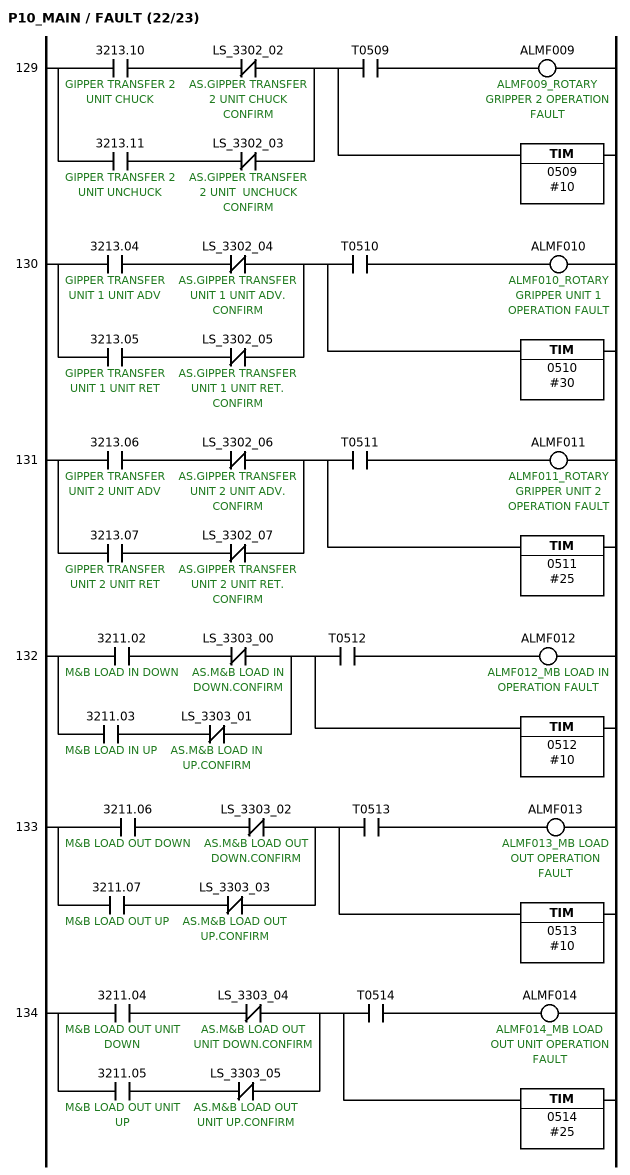
; [picture p24: P10_MAIN / FAULT, rungs 129-134]
; rung 129
LD 3213.10  ; GIPPER TRANSFER 2 UNIT CHUCK
ANDNOT LS_3302_02  ; AS.GIPPER TRANSFER 2 UNIT CHUCK CONFIRM
LD 3213.11  ; GIPPER TRANSFER 2 UNIT UNCHUCK
ANDNOT LS_3302_03  ; AS.GIPPER TRANSFER 2 UNIT  UNCHUCK CONFIRM
ORLD
OUT TR0
AND T0509
OUT ALMF009  ; ALMF009_ROTARY GRIPPER 2 OPERATION FAULT
LD TR0
TIM 0509 #10
; rung 130
LD 3213.04  ; GIPPER TRANSFER UNIT 1 UNIT ADV
ANDNOT LS_3302_04  ; AS.GIPPER TRANSFER UNIT 1 UNIT ADV. CONFIRM
LD 3213.05  ; GIPPER TRANSFER UNIT 1 UNIT RET
ANDNOT LS_3302_05  ; AS.GIPPER TRANSFER UNIT 1 UNIT RET. CONFIRM
ORLD
OUT TR0
AND T0510
OUT ALMF010  ; ALMF010_ROTARY GRIPPER UNIT 1 OPERATION FAULT
LD TR0
TIM 0510 #30
; rung 131
LD 3213.06  ; GIPPER TRANSFER UNIT 2 UNIT ADV
ANDNOT LS_3302_06  ; AS.GIPPER TRANSFER UNIT 2 UNIT ADV. CONFIRM
LD 3213.07  ; GIPPER TRANSFER UNIT 2 UNIT RET
ANDNOT LS_3302_07  ; AS.GIPPER TRANSFER UNIT 2 UNIT RET. CONFIRM
ORLD
OUT TR0
AND T0511
OUT ALMF011  ; ALMF011_ROTARY GRIPPER UNIT 2 OPERATION FAULT
LD TR0
TIM 0511 #25
; rung 132
LD 3211.02  ; M&B LOAD IN DOWN
ANDNOT LS_3303_00  ; AS.M&B LOAD IN DOWN.CONFIRM
LD 3211.03  ; M&B LOAD IN UP
ANDNOT LS_3303_01  ; AS.M&B LOAD IN UP.CONFIRM
ORLD
OUT TR0
AND T0512
OUT ALMF012  ; ALMF012_MB LOAD IN OPERATION FAULT
LD TR0
TIM 0512 #10
; rung 133
LD 3211.06  ; M&B LOAD OUT DOWN
ANDNOT LS_3303_02  ; AS.M&B LOAD OUT DOWN.CONFIRM
LD 3211.07  ; M&B LOAD OUT UP
ANDNOT LS_3303_03  ; AS.M&B LOAD OUT UP.CONFIRM
ORLD
OUT TR0
AND T0513
OUT ALMF013  ; ALMF013_MB LOAD OUT OPERATION FAULT
LD TR0
TIM 0513 #10
; rung 134
LD 3211.04  ; M&B LOAD OUT UNIT DOWN
ANDNOT LS_3303_04  ; AS.M&B LOAD OUT UNIT DOWN.CONFIRM
LD 3211.05  ; M&B LOAD OUT UNIT UP
ANDNOT LS_3303_05  ; AS.M&B LOAD OUT UNIT UP.CONFIRM
ORLD
OUT TR0
AND T0514
OUT ALMF014  ; ALMF014_MB LOAD OUT UNIT OPERATION FAULT
LD TR0
TIM 0514 #25

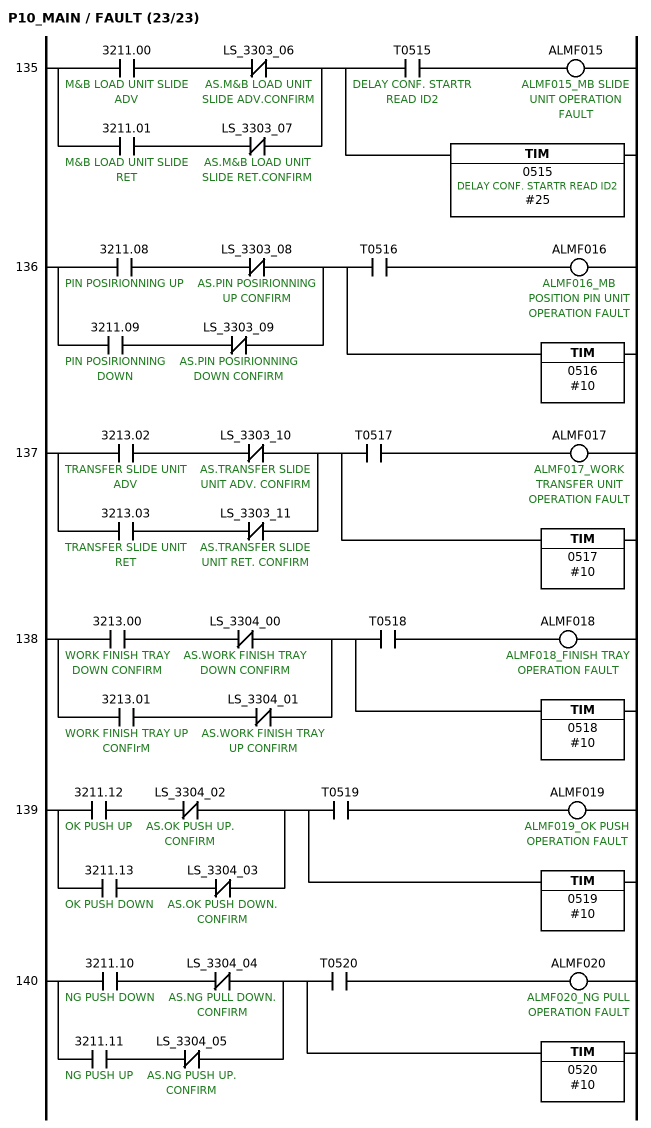
; rung 135
LD 3211.00  ; M&B LOAD UNIT SLIDE ADV
ANDNOT LS_3303_06  ; AS.M&B LOAD UNIT SLIDE ADV.CONFIRM
LD 3211.01  ; M&B LOAD UNIT SLIDE RET
ANDNOT LS_3303_07  ; AS.M&B LOAD UNIT SLIDE RET.CONFIRM
ORLD
OUT TR0
AND T0515  ; DELAY CONF. STARTR READ ID2
OUT ALMF015  ; ALMF015_MB SLIDE UNIT OPERATION FAULT
LD TR0
TIM 0515 #25  ; DELAY CONF. STARTR READ ID2
; rung 136
LD 3211.08  ; PIN POSIRIONNING UP
ANDNOT LS_3303_08  ; AS.PIN POSIRIONNING UP CONFIRM
LD 3211.09  ; PIN POSIRIONNING DOWN
ANDNOT LS_3303_09  ; AS.PIN POSIRIONNING DOWN CONFIRM
ORLD
OUT TR0
AND T0516
OUT ALMF016  ; ALMF016_MB POSITION PIN UNIT OPERATION FAULT
LD TR0
TIM 0516 #10
; rung 137
LD 3213.02  ; TRANSFER SLIDE UNIT ADV
ANDNOT LS_3303_10  ; AS.TRANSFER SLIDE UNIT ADV. CONFIRM
LD 3213.03  ; TRANSFER SLIDE UNIT RET
ANDNOT LS_3303_11  ; AS.TRANSFER SLIDE UNIT RET. CONFIRM
ORLD
OUT TR0
AND T0517
OUT ALMF017  ; ALMF017_WORK TRANSFER UNIT OPERATION FAULT
LD TR0
TIM 0517 #10
; rung 138
LD 3213.00  ; WORK FINISH TRAY DOWN CONFIRM
ANDNOT LS_3304_00  ; AS.WORK FINISH TRAY DOWN CONFIRM
LD 3213.01  ; WORK FINISH TRAY UP CONFIrM
ANDNOT LS_3304_01  ; AS.WORK FINISH TRAY UP CONFIRM
ORLD
OUT TR0
AND T0518
OUT ALMF018  ; ALMF018_FINISH TRAY OPERATION FAULT
LD TR0
TIM 0518 #10
; rung 139
LD 3211.12  ; OK PUSH UP
ANDNOT LS_3304_02  ; AS.OK PUSH UP. CONFIRM
LD 3211.13  ; OK PUSH DOWN
ANDNOT LS_3304_03  ; AS.OK PUSH DOWN. CONFIRM
ORLD
OUT TR0
AND T0519
OUT ALMF019  ; ALMF019_OK PUSH OPERATION FAULT
LD TR0
TIM 0519 #10
; rung 140
LD 3211.10  ; NG PUSH DOWN
ANDNOT LS_3304_04  ; AS.NG PULL DOWN. CONFIRM
LD 3211.11  ; NG PUSH UP
ANDNOT LS_3304_05  ; AS.NG PUSH UP. CONFIRM
ORLD
OUT TR0
AND T0520
OUT ALMF020  ; ALMF020_NG PULL OPERATION FAULT
LD TR0
TIM 0520 #10

### Section INPUT

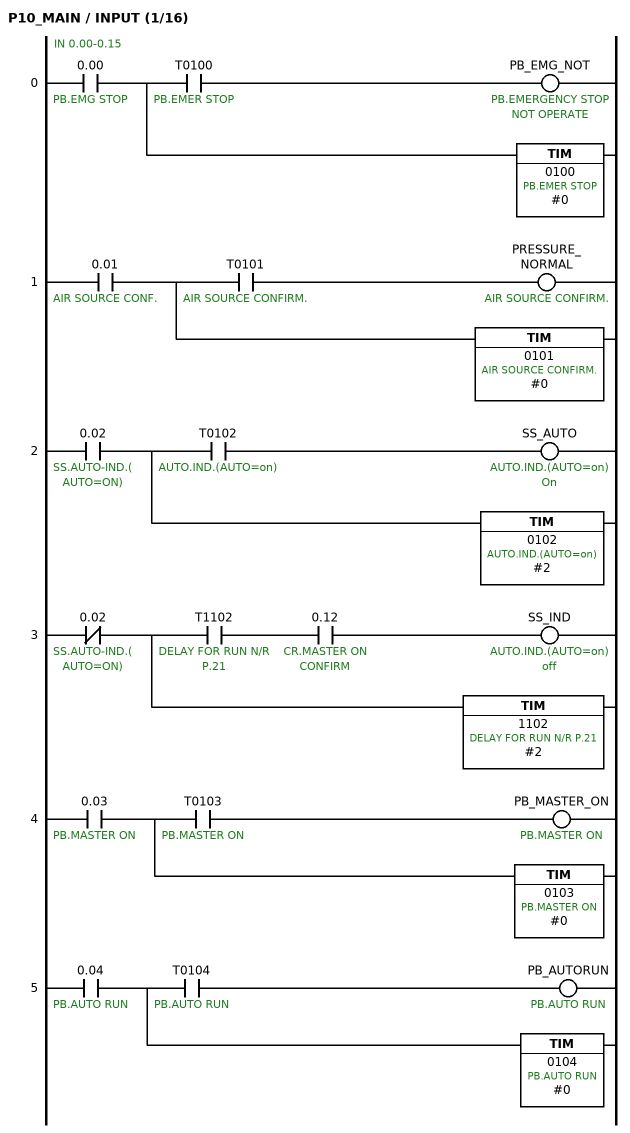
; rung 0: IN 0.00-0.15
LD 0.00  ; PB.EMG STOP
OUT TR0
AND T0100  ; PB.EMER STOP
OUT PB_EMG_NOT  ; PB.EMERGENCY STOP NOT OPERATE
LD TR0
TIM 0100 #0  ; PB.EMER STOP
; rung 1
LD 0.01  ; AIR SOURCE CONF.
OUT TR0
AND T0101  ; AIR SOURCE CONFIRM.
OUT PRESSURE_NORMAL  ; AIR SOURCE CONFIRM.
LD TR0
TIM 0101 #0  ; AIR SOURCE CONFIRM.
; rung 2
LD 0.02  ; SS.AUTO-IND.(AUTO=ON)
OUT TR0
AND T0102  ; AUTO.IND.(AUTO=on)
OUT SS_AUTO  ; AUTO.IND.(AUTO=on) On
LD TR0
TIM 0102 #2  ; AUTO.IND.(AUTO=on)
; rung 3
LDNOT 0.02  ; SS.AUTO-IND.(AUTO=ON)
OUT TR0
AND T1102  ; DELAY FOR RUN N/R P.21
AND 0.12  ; CR.MASTER ON CONFIRM
OUT SS_IND  ; AUTO.IND.(AUTO=on) off
LD TR0
TIM 1102 #2  ; DELAY FOR RUN N/R P.21
; rung 4
LD 0.03  ; PB.MASTER ON
OUT TR0
AND T0103  ; PB.MASTER ON
OUT PB_MASTER_ON  ; PB.MASTER ON
LD TR0
TIM 0103 #0  ; PB.MASTER ON
; rung 5
LD 0.04  ; PB.AUTO RUN
OUT TR0
AND T0104  ; PB.AUTO RUN
OUT PB_AUTORUN  ; PB.AUTO RUN
LD TR0
TIM 0104 #0  ; PB.AUTO RUN

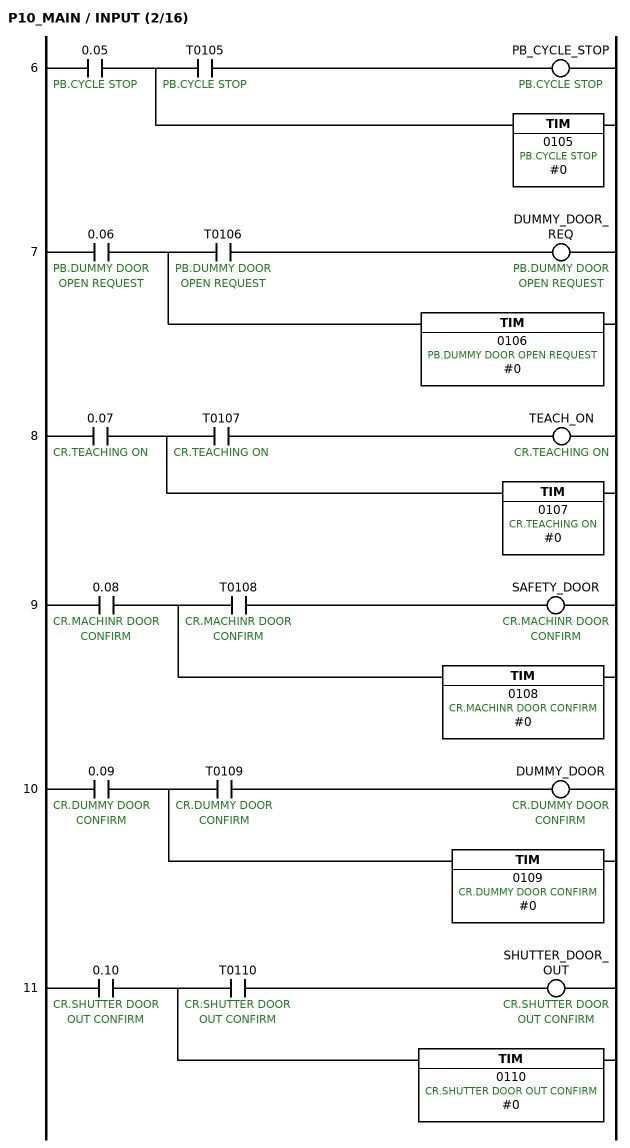
; rung 6
LD 0.05  ; PB.CYCLE STOP
OUT TR0
AND T0105  ; PB.CYCLE STOP
OUT PB_CYCLE_STOP  ; PB.CYCLE STOP
LD TR0
TIM 0105 #0  ; PB.CYCLE STOP
; rung 7
LD 0.06  ; PB.DUMMY DOOR OPEN REQUEST
OUT TR0
AND T0106  ; PB.DUMMY DOOR OPEN REQUEST
OUT DUMMY_DOOR_REQ  ; PB.DUMMY DOOR OPEN REQUEST
LD TR0
TIM 0106 #0  ; PB.DUMMY DOOR OPEN REQUEST
; rung 8
LD 0.07  ; CR.TEACHING ON
OUT TR0
AND T0107  ; CR.TEACHING ON
OUT TEACH_ON  ; CR.TEACHING ON
LD TR0
TIM 0107 #0  ; CR.TEACHING ON
; rung 9
LD 0.08  ; CR.MACHINR DOOR CONFIRM
OUT TR0
AND T0108  ; CR.MACHINR DOOR CONFIRM
OUT SAFETY_DOOR  ; CR.MACHINR DOOR CONFIRM
LD TR0
TIM 0108 #0  ; CR.MACHINR DOOR CONFIRM
; rung 10
LD 0.09  ; CR.DUMMY DOOR CONFIRM
OUT TR0
AND T0109  ; CR.DUMMY DOOR CONFIRM
OUT DUMMY_DOOR  ; CR.DUMMY DOOR CONFIRM
LD TR0
TIM 0109 #0  ; CR.DUMMY DOOR CONFIRM
; rung 11
LD 0.10  ; CR.SHUTTER DOOR OUT CONFIRM
OUT TR0
AND T0110  ; CR.SHUTTER DOOR OUT CONFIRM
OUT SHUTTER_DOOR_OUT  ; CR.SHUTTER DOOR OUT CONFIRM
LD TR0
TIM 0110 #0  ; CR.SHUTTER DOOR OUT CONFIRM

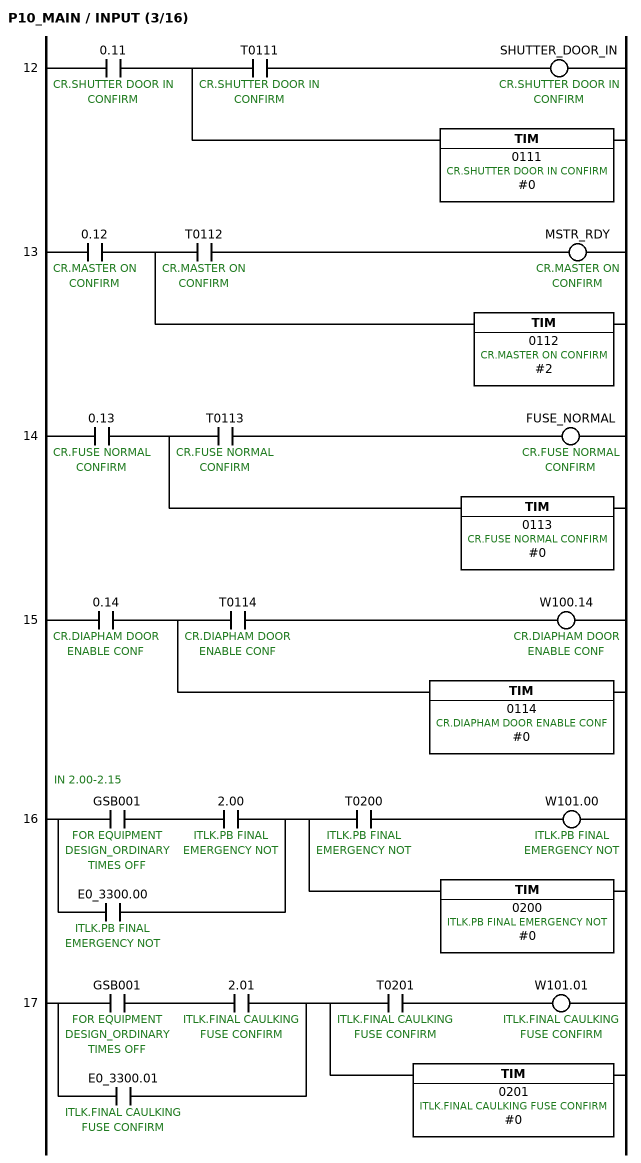
; rung 12
LD 0.11  ; CR.SHUTTER DOOR IN CONFIRM
OUT TR0
AND T0111  ; CR.SHUTTER DOOR IN CONFIRM
OUT SHUTTER_DOOR_IN  ; CR.SHUTTER DOOR IN CONFIRM
LD TR0
TIM 0111 #0  ; CR.SHUTTER DOOR IN CONFIRM
; rung 13
LD 0.12  ; CR.MASTER ON CONFIRM
OUT TR0
AND T0112  ; CR.MASTER ON CONFIRM
OUT MSTR_RDY  ; CR.MASTER ON CONFIRM
LD TR0
TIM 0112 #2  ; CR.MASTER ON CONFIRM
; rung 14
LD 0.13  ; CR.FUSE NORMAL CONFIRM
OUT TR0
AND T0113  ; CR.FUSE NORMAL CONFIRM
OUT FUSE_NORMAL  ; CR.FUSE NORMAL CONFIRM
LD TR0
TIM 0113 #0  ; CR.FUSE NORMAL CONFIRM
; rung 15
LD 0.14  ; CR.DIAPHAM DOOR ENABLE CONF
OUT TR0
AND T0114  ; CR.DIAPHAM DOOR ENABLE CONF
OUT W100.14  ; CR.DIAPHAM DOOR ENABLE CONF
LD TR0
TIM 0114 #0  ; CR.DIAPHAM DOOR ENABLE CONF
; rung 16: IN 2.00-2.15
LD GSB001  ; FOR EQUIPMENT DESIGN_ORDINARY TIMES OFF
AND 2.00  ; ITLK.PB FINAL EMERGENCY NOT
OR E0_3300.00  ; ITLK.PB FINAL EMERGENCY NOT
OUT TR0
AND T0200  ; ITLK.PB FINAL EMERGENCY NOT
OUT W101.00  ; ITLK.PB FINAL EMERGENCY NOT
LD TR0
TIM 0200 #0  ; ITLK.PB FINAL EMERGENCY NOT
; rung 17
LD GSB001  ; FOR EQUIPMENT DESIGN_ORDINARY TIMES OFF
AND 2.01  ; ITLK.FINAL CAULKING FUSE CONFIRM
OR E0_3300.01  ; ITLK.FINAL CAULKING FUSE CONFIRM
OUT TR0
AND T0201  ; ITLK.FINAL CAULKING FUSE CONFIRM
OUT W101.01  ; ITLK.FINAL CAULKING FUSE CONFIRM
LD TR0
TIM 0201 #0  ; ITLK.FINAL CAULKING FUSE CONFIRM

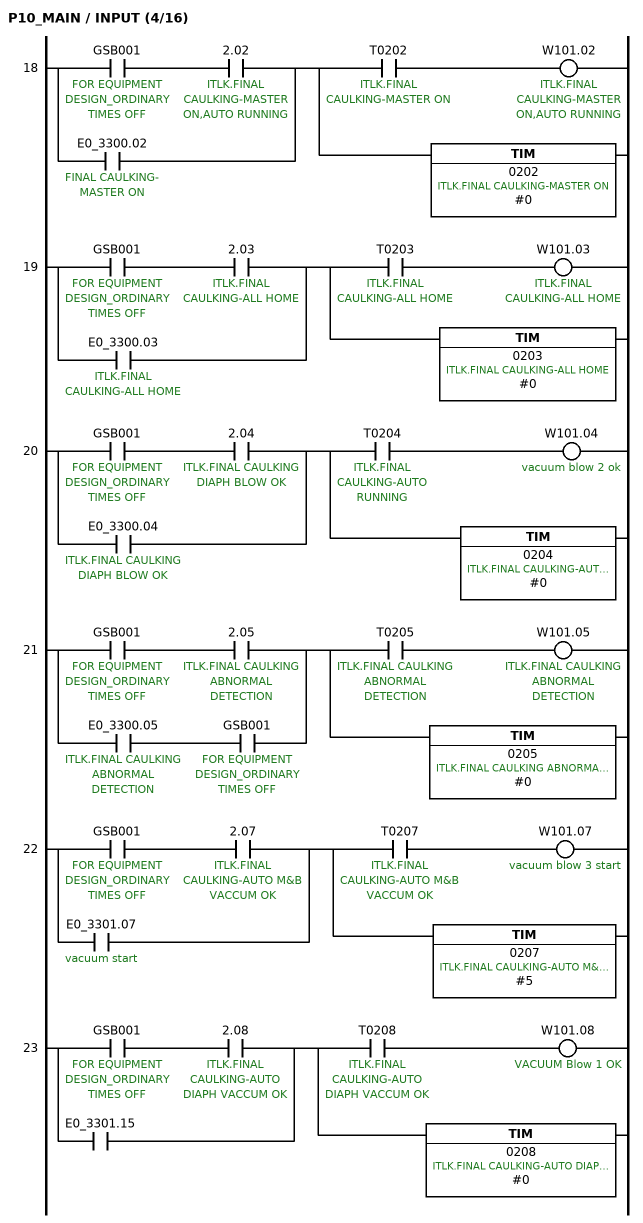
; rung 18
LD GSB001  ; FOR EQUIPMENT DESIGN_ORDINARY TIMES OFF
AND 2.02  ; ITLK.FINAL CAULKING-MASTER ON,AUTO RUNNING
OR E0_3300.02  ; FINAL CAULKING-MASTER ON
OUT TR0
AND T0202  ; ITLK.FINAL CAULKING-MASTER ON
OUT W101.02  ; ITLK.FINAL CAULKING-MASTER ON,AUTO RUNNING
LD TR0
TIM 0202 #0  ; ITLK.FINAL CAULKING-MASTER ON
; rung 19
LD GSB001  ; FOR EQUIPMENT DESIGN_ORDINARY TIMES OFF
AND 2.03  ; ITLK.FINAL CAULKING-ALL HOME
OR E0_3300.03  ; ITLK.FINAL CAULKING-ALL HOME
OUT TR0
AND T0203  ; ITLK.FINAL CAULKING-ALL HOME
OUT W101.03  ; ITLK.FINAL CAULKING-ALL HOME
LD TR0
TIM 0203 #0  ; ITLK.FINAL CAULKING-ALL HOME
; rung 20
LD GSB001  ; FOR EQUIPMENT DESIGN_ORDINARY TIMES OFF
AND 2.04  ; ITLK.FINAL CAULKING DIAPH BLOW OK
OR E0_3300.04  ; ITLK.FINAL CAULKING DIAPH BLOW OK
OUT TR0
AND T0204  ; ITLK.FINAL CAULKING-AUTO RUNNING
OUT W101.04  ; vacuum blow 2 ok
LD TR0
TIM 0204 #0  ; ITLK.FINAL CAULKING-AUTO RUNNING
; rung 21
LD GSB001  ; FOR EQUIPMENT DESIGN_ORDINARY TIMES OFF
AND 2.05  ; ITLK.FINAL CAULKING ABNORMAL DETECTION
LD E0_3300.05  ; ITLK.FINAL CAULKING ABNORMAL DETECTION
AND GSB001  ; FOR EQUIPMENT DESIGN_ORDINARY TIMES OFF
ORLD
OUT TR0
AND T0205  ; ITLK.FINAL CAULKING ABNORMAL DETECTION
OUT W101.05  ; ITLK.FINAL CAULKING ABNORMAL DETECTION
LD TR0
TIM 0205 #0  ; ITLK.FINAL CAULKING ABNORMAL DETECTION
; rung 22
LD GSB001  ; FOR EQUIPMENT DESIGN_ORDINARY TIMES OFF
AND 2.07  ; ITLK.FINAL CAULKING-AUTO M&B VACCUM OK
OR E0_3301.07  ; vacuum start
OUT TR0
AND T0207  ; ITLK.FINAL CAULKING-AUTO M&B VACCUM OK
OUT W101.07  ; vacuum blow 3 start
LD TR0
TIM 0207 #5  ; ITLK.FINAL CAULKING-AUTO M&B VACCUM OK
; rung 23
LD GSB001  ; FOR EQUIPMENT DESIGN_ORDINARY TIMES OFF
AND 2.08  ; ITLK.FINAL CAULKING-AUTO DIAPH VACCUM OK
OR E0_3301.15
OUT TR0
AND T0208  ; ITLK.FINAL CAULKING-AUTO DIAPH VACCUM OK
OUT W101.08  ; VACUUM Blow 1 OK
LD TR0
TIM 0208 #0  ; ITLK.FINAL CAULKING-AUTO DIAPH VACCUM OK

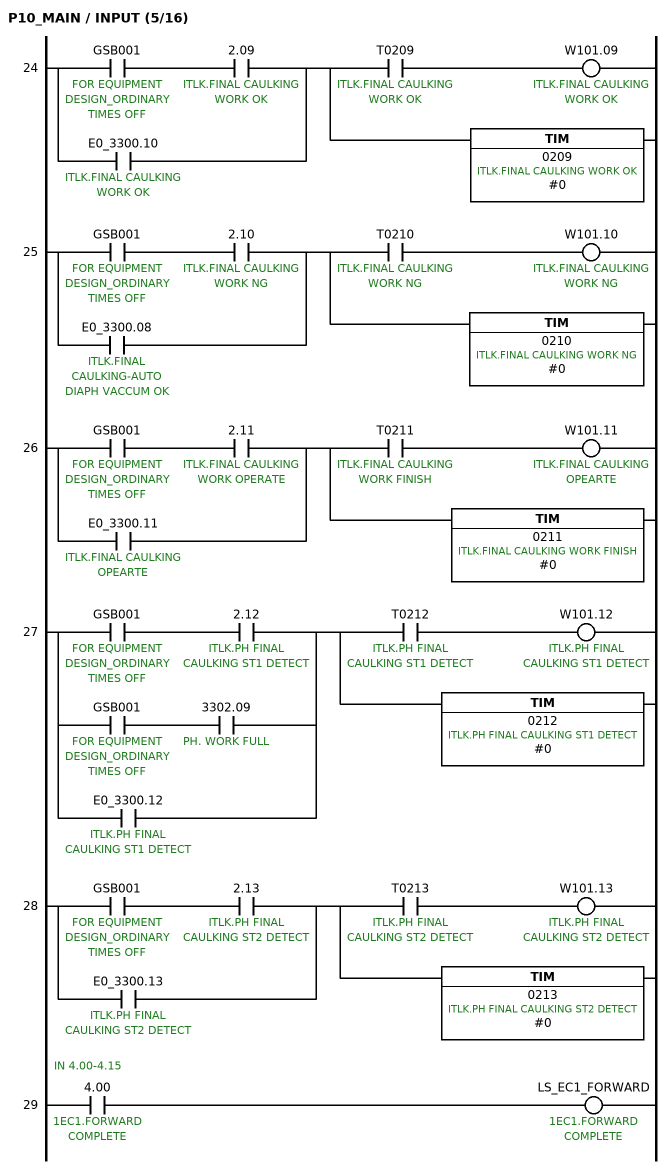
; rung 24
LD GSB001  ; FOR EQUIPMENT DESIGN_ORDINARY TIMES OFF
AND 2.09  ; ITLK.FINAL CAULKING WORK OK
OR E0_3300.10  ; ITLK.FINAL CAULKING WORK OK
OUT TR0
AND T0209  ; ITLK.FINAL CAULKING WORK OK
OUT W101.09  ; ITLK.FINAL CAULKING WORK OK
LD TR0
TIM 0209 #0  ; ITLK.FINAL CAULKING WORK OK
; rung 25
LD GSB001  ; FOR EQUIPMENT DESIGN_ORDINARY TIMES OFF
AND 2.10  ; ITLK.FINAL CAULKING WORK NG
OR E0_3300.08  ; ITLK.FINAL CAULKING-AUTO DIAPH VACCUM OK
OUT TR0
AND T0210  ; ITLK.FINAL CAULKING WORK NG
OUT W101.10  ; ITLK.FINAL CAULKING WORK NG
LD TR0
TIM 0210 #0  ; ITLK.FINAL CAULKING WORK NG
; rung 26
LD GSB001  ; FOR EQUIPMENT DESIGN_ORDINARY TIMES OFF
AND 2.11  ; ITLK.FINAL CAULKING WORK OPERATE
OR E0_3300.11  ; ITLK.FINAL CAULKING OPEARTE
OUT TR0
AND T0211  ; ITLK.FINAL CAULKING WORK FINISH
OUT W101.11  ; ITLK.FINAL CAULKING OPEARTE
LD TR0
TIM 0211 #0  ; ITLK.FINAL CAULKING WORK FINISH
; rung 27
LD GSB001  ; FOR EQUIPMENT DESIGN_ORDINARY TIMES OFF
AND 2.12  ; ITLK.PH FINAL CAULKING ST1 DETECT
LD GSB001  ; FOR EQUIPMENT DESIGN_ORDINARY TIMES OFF
AND 3302.09  ; PH. WORK FULL
ORLD
OR E0_3300.12  ; ITLK.PH FINAL CAULKING ST1 DETECT
OUT TR0
AND T0212  ; ITLK.PH FINAL CAULKING ST1 DETECT
OUT W101.12  ; ITLK.PH FINAL CAULKING ST1 DETECT
LD TR0
TIM 0212 #0  ; ITLK.PH FINAL CAULKING ST1 DETECT
; rung 28
LD GSB001  ; FOR EQUIPMENT DESIGN_ORDINARY TIMES OFF
AND 2.13  ; ITLK.PH FINAL CAULKING ST2 DETECT
OR E0_3300.13  ; ITLK.PH FINAL CAULKING ST2 DETECT
OUT TR0
AND T0213  ; ITLK.PH FINAL CAULKING ST2 DETECT
OUT W101.13  ; ITLK.PH FINAL CAULKING ST2 DETECT
LD TR0
TIM 0213 #0  ; ITLK.PH FINAL CAULKING ST2 DETECT
; rung 29: IN 4.00-4.15
LD 4.00  ; 1EC1.FORWARD COMPLETE
OUT LS_EC1_FORWARD  ; 1EC1.FORWARD COMPLETE

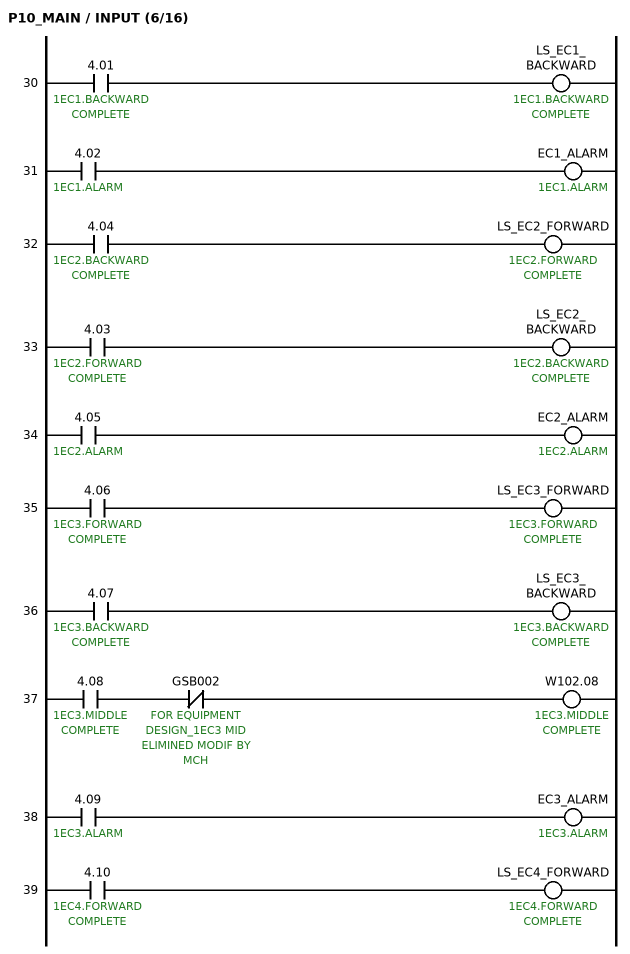
; rung 30
LD 4.01  ; 1EC1.BACKWARD COMPLETE
OUT LS_EC1_BACKWARD  ; 1EC1.BACKWARD COMPLETE
; rung 31
LD 4.02  ; 1EC1.ALARM
OUT EC1_ALARM  ; 1EC1.ALARM
; rung 32
LD 4.04  ; 1EC2.BACKWARD COMPLETE
OUT LS_EC2_FORWARD  ; 1EC2.FORWARD COMPLETE
; rung 33
LD 4.03  ; 1EC2.FORWARD COMPLETE
OUT LS_EC2_BACKWARD  ; 1EC2.BACKWARD COMPLETE
; rung 34
LD 4.05  ; 1EC2.ALARM
OUT EC2_ALARM  ; 1EC2.ALARM
; rung 35
LD 4.06  ; 1EC3.FORWARD COMPLETE
OUT LS_EC3_FORWARD  ; 1EC3.FORWARD COMPLETE
; rung 36
LD 4.07  ; 1EC3.BACKWARD COMPLETE
OUT LS_EC3_BACKWARD  ; 1EC3.BACKWARD COMPLETE
; rung 37
LD 4.08  ; 1EC3.MIDDLE COMPLETE
ANDNOT GSB002  ; FOR EQUIPMENT DESIGN_1EC3 MID ELIMINED MODIF BY MCH
OUT W102.08  ; 1EC3.MIDDLE COMPLETE
; rung 38
LD 4.09  ; 1EC3.ALARM
OUT EC3_ALARM  ; 1EC3.ALARM
; rung 39
LD 4.10  ; 1EC4.FORWARD COMPLETE
OUT LS_EC4_FORWARD  ; 1EC4.FORWARD COMPLETE

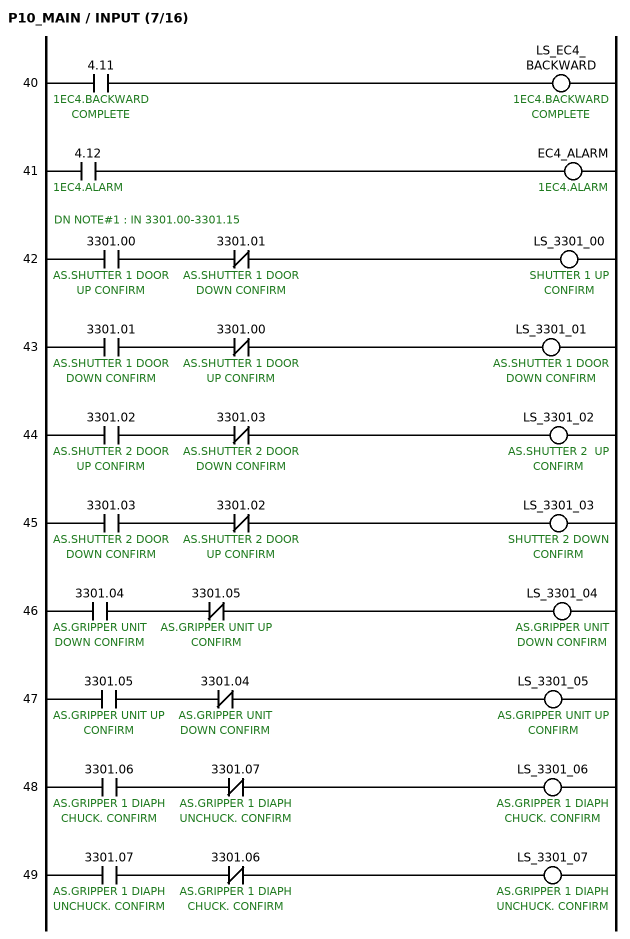
; rung 40
LD 4.11  ; 1EC4.BACKWARD COMPLETE
OUT LS_EC4_BACKWARD  ; 1EC4.BACKWARD COMPLETE
; rung 41
LD 4.12  ; 1EC4.ALARM
OUT EC4_ALARM  ; 1EC4.ALARM
; rung 42: DN NOTE#1 : IN 3301.00-3301.15
LD 3301.00  ; AS.SHUTTER 1 DOOR UP CONFIRM
ANDNOT 3301.01  ; AS.SHUTTER 1 DOOR DOWN CONFIRM
OUT LS_3301_00  ; SHUTTER 1 UP CONFIRM
; rung 43
LD 3301.01  ; AS.SHUTTER 1 DOOR DOWN CONFIRM
ANDNOT 3301.00  ; AS.SHUTTER 1 DOOR UP CONFIRM
OUT LS_3301_01  ; AS.SHUTTER 1 DOOR DOWN CONFIRM
; rung 44
LD 3301.02  ; AS.SHUTTER 2 DOOR UP CONFIRM
ANDNOT 3301.03  ; AS.SHUTTER 2 DOOR DOWN CONFIRM
OUT LS_3301_02  ; AS.SHUTTER 2  UP CONFIRM
; rung 45
LD 3301.03  ; AS.SHUTTER 2 DOOR DOWN CONFIRM
ANDNOT 3301.02  ; AS.SHUTTER 2 DOOR UP CONFIRM
OUT LS_3301_03  ; SHUTTER 2 DOWN CONFIRM
; rung 46
LD 3301.04  ; AS.GRIPPER UNIT DOWN CONFIRM
ANDNOT 3301.05  ; AS.GRIPPER UNIT UP CONFIRM
OUT LS_3301_04  ; AS.GRIPPER UNIT DOWN CONFIRM
; rung 47
LD 3301.05  ; AS.GRIPPER UNIT UP CONFIRM
ANDNOT 3301.04  ; AS.GRIPPER UNIT DOWN CONFIRM
OUT LS_3301_05  ; AS.GRIPPER UNIT UP CONFIRM
; rung 48
LD 3301.06  ; AS.GRIPPER 1 DIAPH CHUCK. CONFIRM
ANDNOT 3301.07  ; AS.GRIPPER 1 DIAPH UNCHUCK. CONFIRM
OUT LS_3301_06  ; AS.GRIPPER 1 DIAPH CHUCK. CONFIRM
; rung 49
LD 3301.07  ; AS.GRIPPER 1 DIAPH UNCHUCK. CONFIRM
ANDNOT 3301.06  ; AS.GRIPPER 1 DIAPH CHUCK. CONFIRM
OUT LS_3301_07  ; AS.GRIPPER 1 DIAPH UNCHUCK. CONFIRM

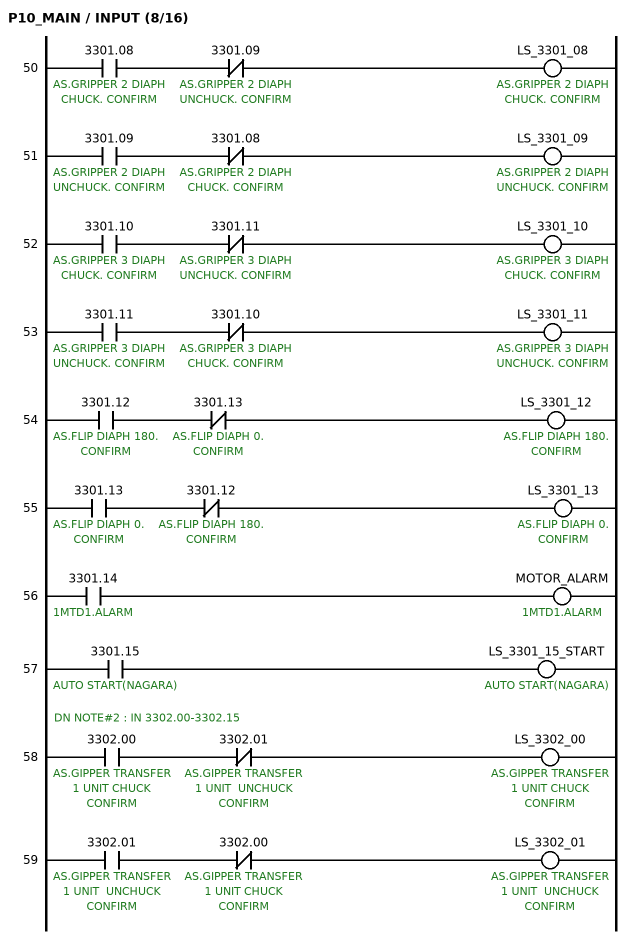
; rung 50
LD 3301.08  ; AS.GRIPPER 2 DIAPH CHUCK. CONFIRM
ANDNOT 3301.09  ; AS.GRIPPER 2 DIAPH UNCHUCK. CONFIRM
OUT LS_3301_08  ; AS.GRIPPER 2 DIAPH CHUCK. CONFIRM
; rung 51
LD 3301.09  ; AS.GRIPPER 2 DIAPH UNCHUCK. CONFIRM
ANDNOT 3301.08  ; AS.GRIPPER 2 DIAPH CHUCK. CONFIRM
OUT LS_3301_09  ; AS.GRIPPER 2 DIAPH UNCHUCK. CONFIRM
; rung 52
LD 3301.10  ; AS.GRIPPER 3 DIAPH CHUCK. CONFIRM
ANDNOT 3301.11  ; AS.GRIPPER 3 DIAPH UNCHUCK. CONFIRM
OUT LS_3301_10  ; AS.GRIPPER 3 DIAPH CHUCK. CONFIRM
; rung 53
LD 3301.11  ; AS.GRIPPER 3 DIAPH UNCHUCK. CONFIRM
ANDNOT 3301.10  ; AS.GRIPPER 3 DIAPH CHUCK. CONFIRM
OUT LS_3301_11  ; AS.GRIPPER 3 DIAPH UNCHUCK. CONFIRM
; rung 54
LD 3301.12  ; AS.FLIP DIAPH 180. CONFIRM
ANDNOT 3301.13  ; AS.FLIP DIAPH 0. CONFIRM
OUT LS_3301_12  ; AS.FLIP DIAPH 180. CONFIRM
; rung 55
LD 3301.13  ; AS.FLIP DIAPH 0. CONFIRM
ANDNOT 3301.12  ; AS.FLIP DIAPH 180. CONFIRM
OUT LS_3301_13  ; AS.FLIP DIAPH 0. CONFIRM
; rung 56
LD 3301.14  ; 1MTD1.ALARM
OUT MOTOR_ALARM  ; 1MTD1.ALARM
; rung 57
LD 3301.15  ; AUTO START(NAGARA)
OUT LS_3301_15_START  ; AUTO START(NAGARA)
; rung 58: DN NOTE#2 : IN 3302.00-3302.15
LD 3302.00  ; AS.GIPPER TRANSFER 1 UNIT CHUCK CONFIRM
ANDNOT 3302.01  ; AS.GIPPER TRANSFER 1 UNIT  UNCHUCK CONFIRM
OUT LS_3302_00  ; AS.GIPPER TRANSFER 1 UNIT CHUCK CONFIRM
; rung 59
LD 3302.01  ; AS.GIPPER TRANSFER 1 UNIT  UNCHUCK CONFIRM
ANDNOT 3302.00  ; AS.GIPPER TRANSFER 1 UNIT CHUCK CONFIRM
OUT LS_3302_01  ; AS.GIPPER TRANSFER 1 UNIT  UNCHUCK CONFIRM

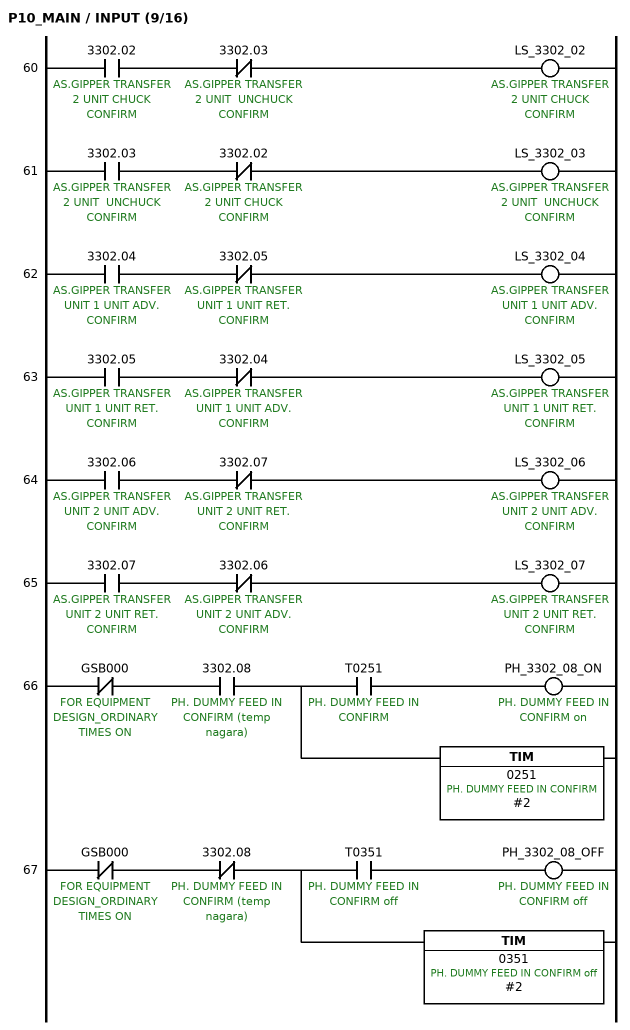
; rung 60
LD 3302.02  ; AS.GIPPER TRANSFER 2 UNIT CHUCK CONFIRM
ANDNOT 3302.03  ; AS.GIPPER TRANSFER 2 UNIT  UNCHUCK CONFIRM
OUT LS_3302_02  ; AS.GIPPER TRANSFER 2 UNIT CHUCK CONFIRM
; rung 61
LD 3302.03  ; AS.GIPPER TRANSFER 2 UNIT  UNCHUCK CONFIRM
ANDNOT 3302.02  ; AS.GIPPER TRANSFER 2 UNIT CHUCK CONFIRM
OUT LS_3302_03  ; AS.GIPPER TRANSFER 2 UNIT  UNCHUCK CONFIRM
; rung 62
LD 3302.04  ; AS.GIPPER TRANSFER UNIT 1 UNIT ADV. CONFIRM
ANDNOT 3302.05  ; AS.GIPPER TRANSFER UNIT 1 UNIT RET. CONFIRM
OUT LS_3302_04  ; AS.GIPPER TRANSFER UNIT 1 UNIT ADV. CONFIRM
; rung 63
LD 3302.05  ; AS.GIPPER TRANSFER UNIT 1 UNIT RET. CONFIRM
ANDNOT 3302.04  ; AS.GIPPER TRANSFER UNIT 1 UNIT ADV. CONFIRM
OUT LS_3302_05  ; AS.GIPPER TRANSFER UNIT 1 UNIT RET. CONFIRM
; rung 64
LD 3302.06  ; AS.GIPPER TRANSFER UNIT 2 UNIT ADV. CONFIRM
ANDNOT 3302.07  ; AS.GIPPER TRANSFER UNIT 2 UNIT RET. CONFIRM
OUT LS_3302_06  ; AS.GIPPER TRANSFER UNIT 2 UNIT ADV. CONFIRM
; rung 65
LD 3302.07  ; AS.GIPPER TRANSFER UNIT 2 UNIT RET. CONFIRM
ANDNOT 3302.06  ; AS.GIPPER TRANSFER UNIT 2 UNIT ADV. CONFIRM
OUT LS_3302_07  ; AS.GIPPER TRANSFER UNIT 2 UNIT RET. CONFIRM
; rung 66
LDNOT GSB000  ; FOR EQUIPMENT DESIGN_ORDINARY TIMES ON
AND 3302.08  ; PH. DUMMY FEED IN CONFIRM (temp nagara)
OUT TR0
AND T0251  ; PH. DUMMY FEED IN CONFIRM
OUT PH_3302_08_ON  ; PH. DUMMY FEED IN CONFIRM on
LD TR0
TIM 0251 #2  ; PH. DUMMY FEED IN CONFIRM
; rung 67
LDNOT GSB000  ; FOR EQUIPMENT DESIGN_ORDINARY TIMES ON
ANDNOT 3302.08  ; PH. DUMMY FEED IN CONFIRM (temp nagara)
OUT TR0
AND T0351  ; PH. DUMMY FEED IN CONFIRM off
OUT PH_3302_08_OFF  ; PH. DUMMY FEED IN CONFIRM off
LD TR0
TIM 0351 #2  ; PH. DUMMY FEED IN CONFIRM off

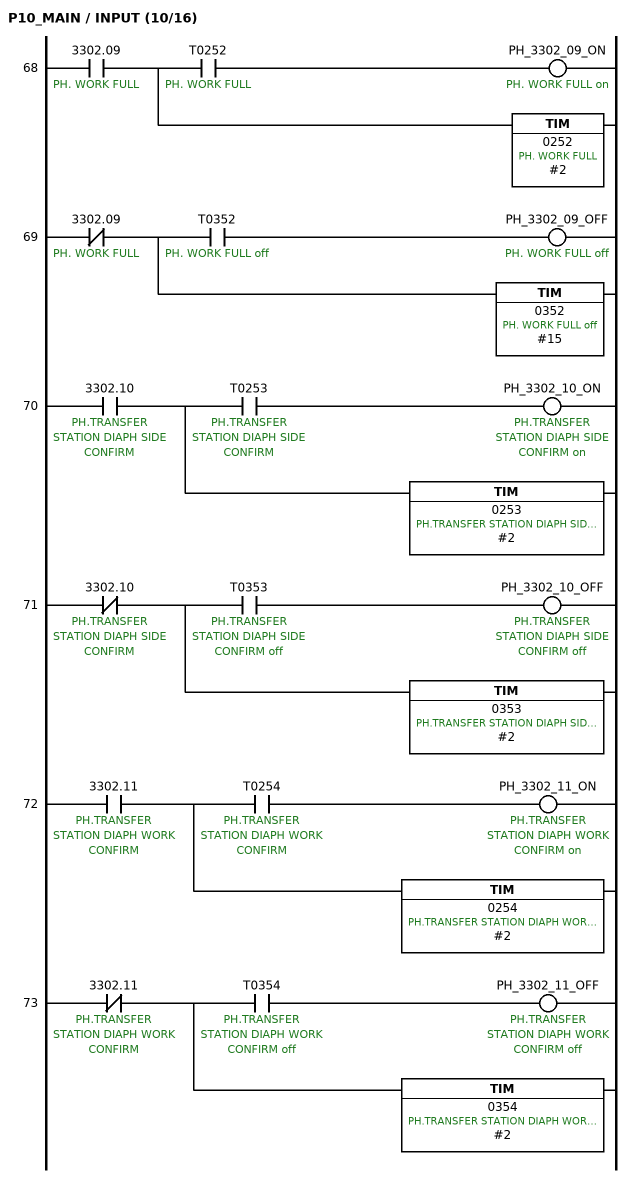
; rung 68
LD 3302.09  ; PH. WORK FULL
OUT TR0
AND T0252  ; PH. WORK FULL
OUT PH_3302_09_ON  ; PH. WORK FULL on
LD TR0
TIM 0252 #2  ; PH. WORK FULL
; rung 69
LDNOT 3302.09  ; PH. WORK FULL
OUT TR0
AND T0352  ; PH. WORK FULL off
OUT PH_3302_09_OFF  ; PH. WORK FULL off
LD TR0
TIM 0352 #15  ; PH. WORK FULL off
; rung 70
LD 3302.10  ; PH.TRANSFER STATION DIAPH SIDE CONFIRM
OUT TR0
AND T0253  ; PH.TRANSFER STATION DIAPH SIDE CONFIRM
OUT PH_3302_10_ON  ; PH.TRANSFER STATION DIAPH SIDE CONFIRM on
LD TR0
TIM 0253 #2  ; PH.TRANSFER STATION DIAPH SIDE CONFIRM
; rung 71
LDNOT 3302.10  ; PH.TRANSFER STATION DIAPH SIDE CONFIRM
OUT TR0
AND T0353  ; PH.TRANSFER STATION DIAPH SIDE CONFIRM off
OUT PH_3302_10_OFF  ; PH.TRANSFER STATION DIAPH SIDE CONFIRM off
LD TR0
TIM 0353 #2  ; PH.TRANSFER STATION DIAPH SIDE CONFIRM off
; rung 72
LD 3302.11  ; PH.TRANSFER STATION DIAPH WORK CONFIRM
OUT TR0
AND T0254  ; PH.TRANSFER STATION DIAPH WORK CONFIRM
OUT PH_3302_11_ON  ; PH.TRANSFER STATION DIAPH WORK CONFIRM on
LD TR0
TIM 0254 #2  ; PH.TRANSFER STATION DIAPH WORK CONFIRM
; rung 73
LDNOT 3302.11  ; PH.TRANSFER STATION DIAPH WORK CONFIRM
OUT TR0
AND T0354  ; PH.TRANSFER STATION DIAPH WORK CONFIRM off
OUT PH_3302_11_OFF  ; PH.TRANSFER STATION DIAPH WORK CONFIRM off
LD TR0
TIM 0354 #2  ; PH.TRANSFER STATION DIAPH WORK CONFIRM off

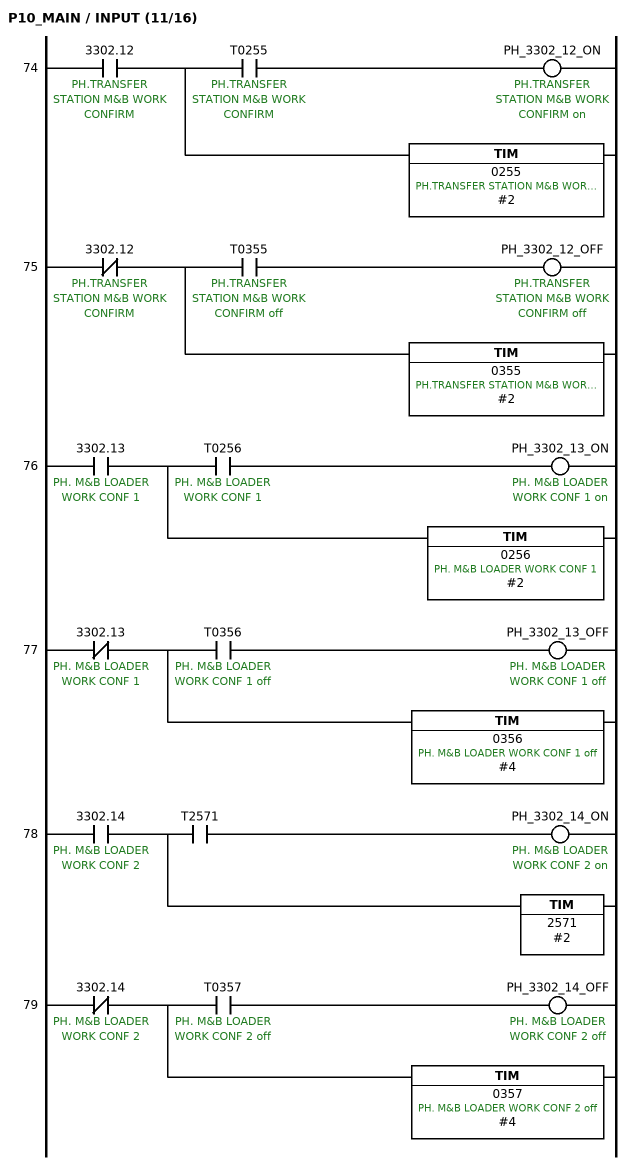
; rung 74
LD 3302.12  ; PH.TRANSFER STATION M&B WORK CONFIRM
OUT TR0
AND T0255  ; PH.TRANSFER STATION M&B WORK CONFIRM
OUT PH_3302_12_ON  ; PH.TRANSFER STATION M&B WORK CONFIRM on
LD TR0
TIM 0255 #2  ; PH.TRANSFER STATION M&B WORK CONFIRM
; rung 75
LDNOT 3302.12  ; PH.TRANSFER STATION M&B WORK CONFIRM
OUT TR0
AND T0355  ; PH.TRANSFER STATION M&B WORK CONFIRM off
OUT PH_3302_12_OFF  ; PH.TRANSFER STATION M&B WORK CONFIRM off
LD TR0
TIM 0355 #2  ; PH.TRANSFER STATION M&B WORK CONFIRM off
; rung 76
LD 3302.13  ; PH. M&B LOADER WORK CONF 1
OUT TR0
AND T0256  ; PH. M&B LOADER WORK CONF 1
OUT PH_3302_13_ON  ; PH. M&B LOADER WORK CONF 1 on
LD TR0
TIM 0256 #2  ; PH. M&B LOADER WORK CONF 1
; rung 77
LDNOT 3302.13  ; PH. M&B LOADER WORK CONF 1
OUT TR0
AND T0356  ; PH. M&B LOADER WORK CONF 1 off
OUT PH_3302_13_OFF  ; PH. M&B LOADER WORK CONF 1 off
LD TR0
TIM 0356 #4  ; PH. M&B LOADER WORK CONF 1 off
; rung 78
LD 3302.14  ; PH. M&B LOADER WORK CONF 2
OUT TR0
AND T2571
OUT PH_3302_14_ON  ; PH. M&B LOADER WORK CONF 2 on
LD TR0
TIM 2571 #2
; rung 79
LDNOT 3302.14  ; PH. M&B LOADER WORK CONF 2
OUT TR0
AND T0357  ; PH. M&B LOADER WORK CONF 2 off
OUT PH_3302_14_OFF  ; PH. M&B LOADER WORK CONF 2 off
LD TR0
TIM 0357 #4  ; PH. M&B LOADER WORK CONF 2 off

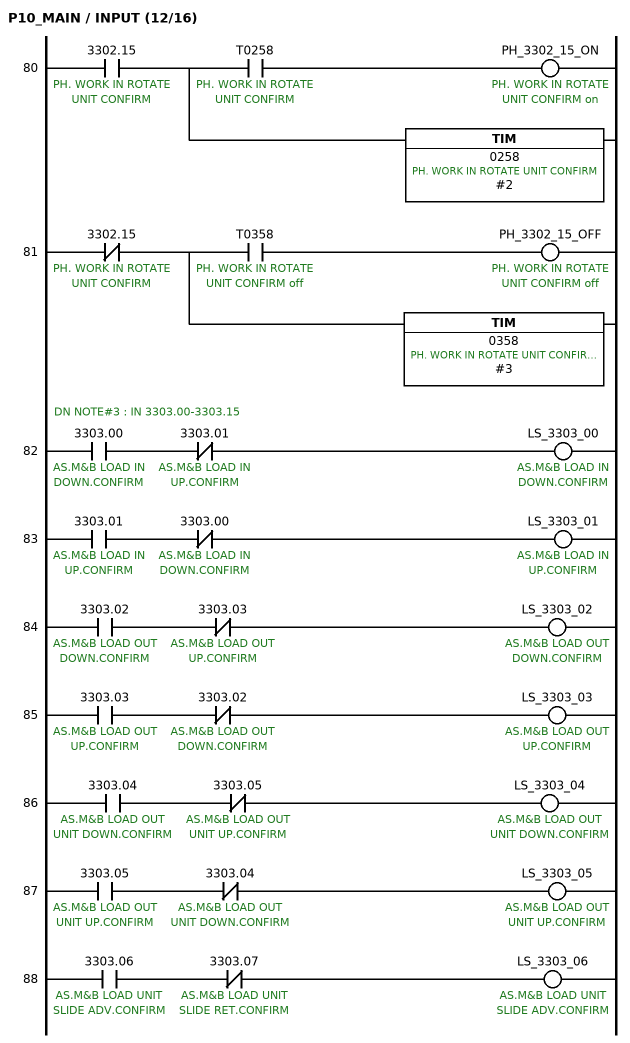
; rung 80
LD 3302.15  ; PH. WORK IN ROTATE UNIT CONFIRM
OUT TR0
AND T0258  ; PH. WORK IN ROTATE UNIT CONFIRM
OUT PH_3302_15_ON  ; PH. WORK IN ROTATE UNIT CONFIRM on
LD TR0
TIM 0258 #2  ; PH. WORK IN ROTATE UNIT CONFIRM
; rung 81
LDNOT 3302.15  ; PH. WORK IN ROTATE UNIT CONFIRM
OUT TR0
AND T0358  ; PH. WORK IN ROTATE UNIT CONFIRM off
OUT PH_3302_15_OFF  ; PH. WORK IN ROTATE UNIT CONFIRM off
LD TR0
TIM 0358 #3  ; PH. WORK IN ROTATE UNIT CONFIRM off
; rung 82: DN NOTE#3 : IN 3303.00-3303.15
LD 3303.00  ; AS.M&B LOAD IN DOWN.CONFIRM
ANDNOT 3303.01  ; AS.M&B LOAD IN UP.CONFIRM
OUT LS_3303_00  ; AS.M&B LOAD IN DOWN.CONFIRM
; rung 83
LD 3303.01  ; AS.M&B LOAD IN UP.CONFIRM
ANDNOT 3303.00  ; AS.M&B LOAD IN DOWN.CONFIRM
OUT LS_3303_01  ; AS.M&B LOAD IN UP.CONFIRM
; rung 84
LD 3303.02  ; AS.M&B LOAD OUT DOWN.CONFIRM
ANDNOT 3303.03  ; AS.M&B LOAD OUT UP.CONFIRM
OUT LS_3303_02  ; AS.M&B LOAD OUT DOWN.CONFIRM
; rung 85
LD 3303.03  ; AS.M&B LOAD OUT UP.CONFIRM
ANDNOT 3303.02  ; AS.M&B LOAD OUT DOWN.CONFIRM
OUT LS_3303_03  ; AS.M&B LOAD OUT UP.CONFIRM
; rung 86
LD 3303.04  ; AS.M&B LOAD OUT UNIT DOWN.CONFIRM
ANDNOT 3303.05  ; AS.M&B LOAD OUT UNIT UP.CONFIRM
OUT LS_3303_04  ; AS.M&B LOAD OUT UNIT DOWN.CONFIRM
; rung 87
LD 3303.05  ; AS.M&B LOAD OUT UNIT UP.CONFIRM
ANDNOT 3303.04  ; AS.M&B LOAD OUT UNIT DOWN.CONFIRM
OUT LS_3303_05  ; AS.M&B LOAD OUT UNIT UP.CONFIRM
; rung 88
LD 3303.06  ; AS.M&B LOAD UNIT SLIDE ADV.CONFIRM
ANDNOT 3303.07  ; AS.M&B LOAD UNIT SLIDE RET.CONFIRM
OUT LS_3303_06  ; AS.M&B LOAD UNIT SLIDE ADV.CONFIRM

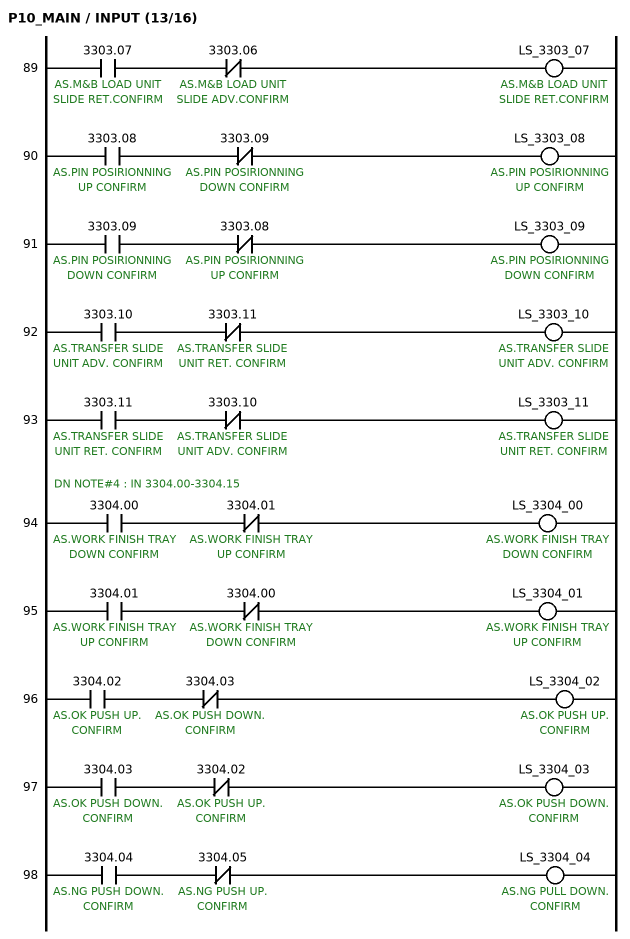
; rung 89
LD 3303.07  ; AS.M&B LOAD UNIT SLIDE RET.CONFIRM
ANDNOT 3303.06  ; AS.M&B LOAD UNIT SLIDE ADV.CONFIRM
OUT LS_3303_07  ; AS.M&B LOAD UNIT SLIDE RET.CONFIRM
; rung 90
LD 3303.08  ; AS.PIN POSIRIONNING UP CONFIRM
ANDNOT 3303.09  ; AS.PIN POSIRIONNING DOWN CONFIRM
OUT LS_3303_08  ; AS.PIN POSIRIONNING UP CONFIRM
; rung 91
LD 3303.09  ; AS.PIN POSIRIONNING DOWN CONFIRM
ANDNOT 3303.08  ; AS.PIN POSIRIONNING UP CONFIRM
OUT LS_3303_09  ; AS.PIN POSIRIONNING DOWN CONFIRM
; rung 92
LD 3303.10  ; AS.TRANSFER SLIDE UNIT ADV. CONFIRM
ANDNOT 3303.11  ; AS.TRANSFER SLIDE UNIT RET. CONFIRM
OUT LS_3303_10  ; AS.TRANSFER SLIDE UNIT ADV. CONFIRM
; rung 93
LD 3303.11  ; AS.TRANSFER SLIDE UNIT RET. CONFIRM
ANDNOT 3303.10  ; AS.TRANSFER SLIDE UNIT ADV. CONFIRM
OUT LS_3303_11  ; AS.TRANSFER SLIDE UNIT RET. CONFIRM
; rung 94: DN NOTE#4 : IN 3304.00-3304.15
LD 3304.00  ; AS.WORK FINISH TRAY DOWN CONFIRM
ANDNOT 3304.01  ; AS.WORK FINISH TRAY UP CONFIRM
OUT LS_3304_00  ; AS.WORK FINISH TRAY DOWN CONFIRM
; rung 95
LD 3304.01  ; AS.WORK FINISH TRAY UP CONFIRM
ANDNOT 3304.00  ; AS.WORK FINISH TRAY DOWN CONFIRM
OUT LS_3304_01  ; AS.WORK FINISH TRAY UP CONFIRM
; rung 96
LD 3304.02  ; AS.OK PUSH UP. CONFIRM
ANDNOT 3304.03  ; AS.OK PUSH DOWN. CONFIRM
OUT LS_3304_02  ; AS.OK PUSH UP. CONFIRM
; rung 97
LD 3304.03  ; AS.OK PUSH DOWN. CONFIRM
ANDNOT 3304.02  ; AS.OK PUSH UP. CONFIRM
OUT LS_3304_03  ; AS.OK PUSH DOWN. CONFIRM
; rung 98
LD 3304.04  ; AS.NG PUSH DOWN. CONFIRM
ANDNOT 3304.05  ; AS.NG PUSH UP. CONFIRM
OUT LS_3304_04  ; AS.NG PULL DOWN. CONFIRM

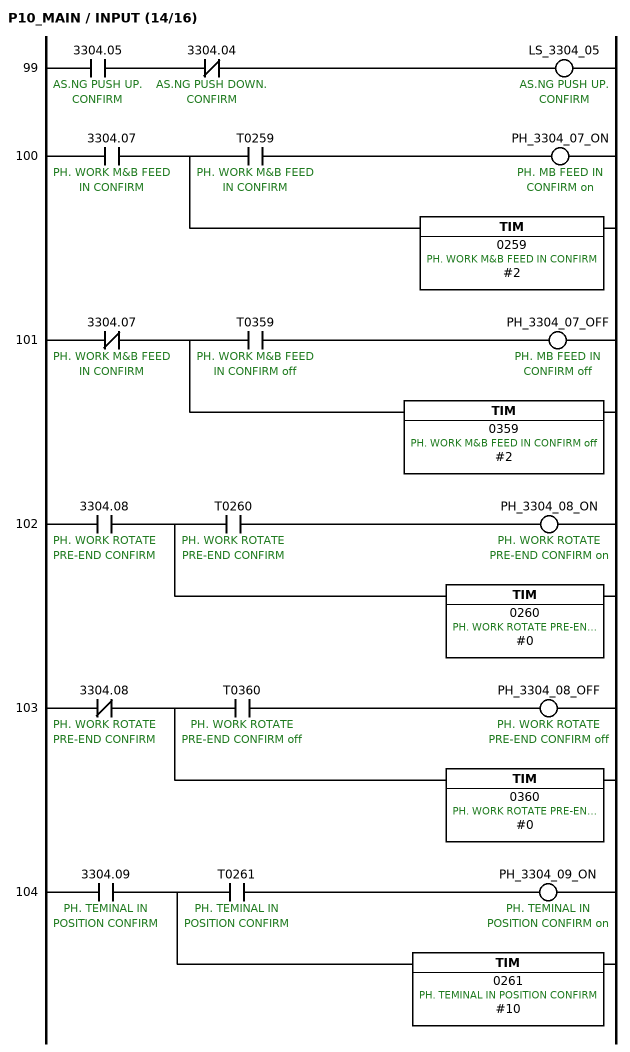
; rung 99
LD 3304.05  ; AS.NG PUSH UP. CONFIRM
ANDNOT 3304.04  ; AS.NG PUSH DOWN. CONFIRM
OUT LS_3304_05  ; AS.NG PUSH UP. CONFIRM
; rung 100
LD 3304.07  ; PH. WORK M&B FEED IN CONFIRM
OUT TR0
AND T0259  ; PH. WORK M&B FEED IN CONFIRM
OUT PH_3304_07_ON  ; PH. MB FEED IN CONFIRM on
LD TR0
TIM 0259 #2  ; PH. WORK M&B FEED IN CONFIRM
; rung 101
LDNOT 3304.07  ; PH. WORK M&B FEED IN CONFIRM
OUT TR0
AND T0359  ; PH. WORK M&B FEED IN CONFIRM off
OUT PH_3304_07_OFF  ; PH. MB FEED IN CONFIRM off
LD TR0
TIM 0359 #2  ; PH. WORK M&B FEED IN CONFIRM off
; rung 102
LD 3304.08  ; PH. WORK ROTATE PRE-END CONFIRM
OUT TR0
AND T0260  ; PH. WORK ROTATE PRE-END CONFIRM
OUT PH_3304_08_ON  ; PH. WORK ROTATE PRE-END CONFIRM on
LD TR0
TIM 0260 #0  ; PH. WORK ROTATE PRE-END CONFIRM
; rung 103
LDNOT 3304.08  ; PH. WORK ROTATE PRE-END CONFIRM
OUT TR0
AND T0360  ; PH. WORK ROTATE PRE-END CONFIRM off
OUT PH_3304_08_OFF  ; PH. WORK ROTATE PRE-END CONFIRM off
LD TR0
TIM 0360 #0  ; PH. WORK ROTATE PRE-END CONFIRM off
; rung 104
LD 3304.09  ; PH. TEMINAL IN POSITION CONFIRM
OUT TR0
AND T0261  ; PH. TEMINAL IN POSITION CONFIRM
OUT PH_3304_09_ON  ; PH. TEMINAL IN POSITION CONFIRM on
LD TR0
TIM 0261 #10  ; PH. TEMINAL IN POSITION CONFIRM

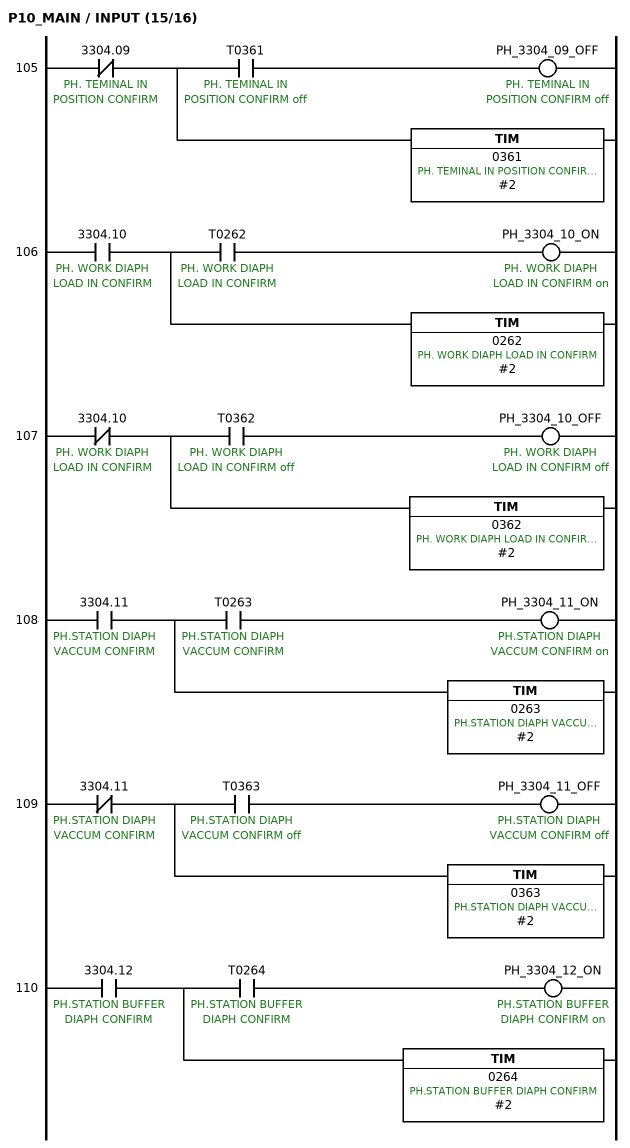
; rung 105
LDNOT 3304.09  ; PH. TEMINAL IN POSITION CONFIRM
OUT TR0
AND T0361  ; PH. TEMINAL IN POSITION CONFIRM off
OUT PH_3304_09_OFF  ; PH. TEMINAL IN POSITION CONFIRM off
LD TR0
TIM 0361 #2  ; PH. TEMINAL IN POSITION CONFIRM off
; rung 106
LD 3304.10  ; PH. WORK DIAPH LOAD IN CONFIRM
OUT TR0
AND T0262  ; PH. WORK DIAPH LOAD IN CONFIRM
OUT PH_3304_10_ON  ; PH. WORK DIAPH LOAD IN CONFIRM on
LD TR0
TIM 0262 #2  ; PH. WORK DIAPH LOAD IN CONFIRM
; rung 107
LDNOT 3304.10  ; PH. WORK DIAPH LOAD IN CONFIRM
OUT TR0
AND T0362  ; PH. WORK DIAPH LOAD IN CONFIRM off
OUT PH_3304_10_OFF  ; PH. WORK DIAPH LOAD IN CONFIRM off
LD TR0
TIM 0362 #2  ; PH. WORK DIAPH LOAD IN CONFIRM off
; rung 108
LD 3304.11  ; PH.STATION DIAPH VACCUM CONFIRM
OUT TR0
AND T0263  ; PH.STATION DIAPH VACCUM CONFIRM
OUT PH_3304_11_ON  ; PH.STATION DIAPH VACCUM CONFIRM on
LD TR0
TIM 0263 #2  ; PH.STATION DIAPH VACCUM CONFIRM
; rung 109
LDNOT 3304.11  ; PH.STATION DIAPH VACCUM CONFIRM
OUT TR0
AND T0363  ; PH.STATION DIAPH VACCUM CONFIRM off
OUT PH_3304_11_OFF  ; PH.STATION DIAPH VACCUM CONFIRM off
LD TR0
TIM 0363 #2  ; PH.STATION DIAPH VACCUM CONFIRM off
; rung 110
LD 3304.12  ; PH.STATION BUFFER DIAPH CONFIRM
OUT TR0
AND T0264  ; PH.STATION BUFFER DIAPH CONFIRM
OUT PH_3304_12_ON  ; PH.STATION BUFFER DIAPH CONFIRM on
LD TR0
TIM 0264 #2  ; PH.STATION BUFFER DIAPH CONFIRM

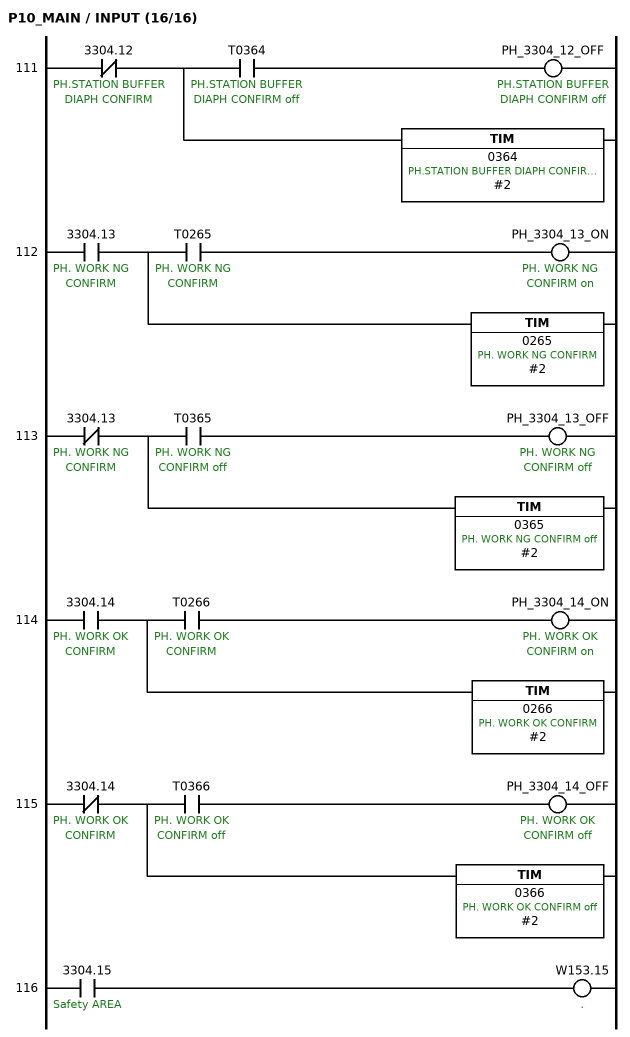
; rung 111
LDNOT 3304.12  ; PH.STATION BUFFER DIAPH CONFIRM
OUT TR0
AND T0364  ; PH.STATION BUFFER DIAPH CONFIRM off
OUT PH_3304_12_OFF  ; PH.STATION BUFFER DIAPH CONFIRM off
LD TR0
TIM 0364 #2  ; PH.STATION BUFFER DIAPH CONFIRM off
; rung 112
LD 3304.13  ; PH. WORK NG CONFIRM
OUT TR0
AND T0265  ; PH. WORK NG CONFIRM
OUT PH_3304_13_ON  ; PH. WORK NG CONFIRM on
LD TR0
TIM 0265 #2  ; PH. WORK NG CONFIRM
; rung 113
LDNOT 3304.13  ; PH. WORK NG CONFIRM
OUT TR0
AND T0365  ; PH. WORK NG CONFIRM off
OUT PH_3304_13_OFF  ; PH. WORK NG CONFIRM off
LD TR0
TIM 0365 #2  ; PH. WORK NG CONFIRM off
; rung 114
LD 3304.14  ; PH. WORK OK CONFIRM
OUT TR0
AND T0266  ; PH. WORK OK CONFIRM
OUT PH_3304_14_ON  ; PH. WORK OK CONFIRM on
LD TR0
TIM 0266 #2  ; PH. WORK OK CONFIRM
; rung 115
LDNOT 3304.14  ; PH. WORK OK CONFIRM
OUT TR0
AND T0366  ; PH. WORK OK CONFIRM off
OUT PH_3304_14_OFF  ; PH. WORK OK CONFIRM off
LD TR0
TIM 0366 #2  ; PH. WORK OK CONFIRM off
; rung 116
LD 3304.15  ; Safety AREA
OUT W153.15  ; .

### Section Device_Output

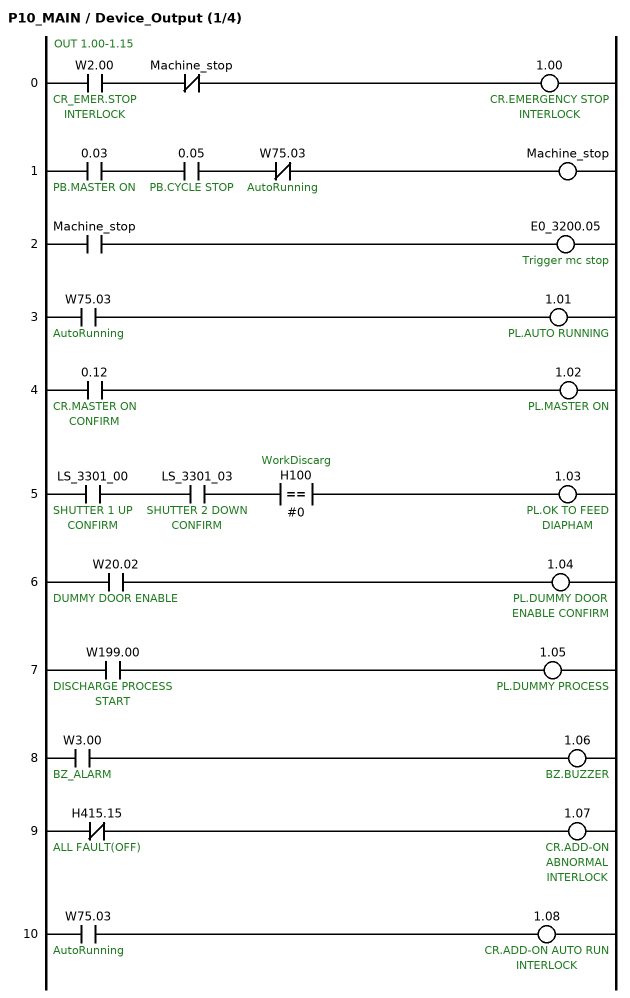
; rung 0: OUT 1.00-1.15
LD W2.00  ; CR_EMER.STOP INTERLOCK
ANDNOT Machine_stop
OUT 1.00  ; CR.EMERGENCY STOP INTERLOCK
; rung 1
LD 0.03  ; PB.MASTER ON
AND 0.05  ; PB.CYCLE STOP
ANDNOT W75.03  ; AutoRunning
OUT Machine_stop
; rung 2
LD Machine_stop
OUT E0_3200.05  ; Trigger mc stop
; rung 3
LD W75.03  ; AutoRunning
OUT 1.01  ; PL.AUTO RUNNING
; rung 4
LD 0.12  ; CR.MASTER ON CONFIRM
OUT 1.02  ; PL.MASTER ON
; rung 5
LD LS_3301_00  ; SHUTTER 1 UP CONFIRM
AND LS_3301_03  ; SHUTTER 2 DOWN CONFIRM
AND=(300) H100 #0  ; WorkDiscarg
OUT 1.03  ; PL.OK TO FEED DIAPHAM
; rung 6
LD W20.02  ; DUMMY DOOR ENABLE
OUT 1.04  ; PL.DUMMY DOOR ENABLE CONFIRM
; rung 7
LD W199.00  ; DISCHARGE PROCESS START
OUT 1.05  ; PL.DUMMY PROCESS
; rung 8
LD W3.00  ; BZ_ALARM
OUT 1.06  ; BZ.BUZZER
; rung 9
LDNOT H415.15  ; ALL FAULT(OFF)
OUT 1.07  ; CR.ADD-ON ABNORMAL INTERLOCK
; rung 10
LD W75.03  ; AutoRunning
OUT 1.08  ; CR.ADD-ON AUTO RUN INTERLOCK

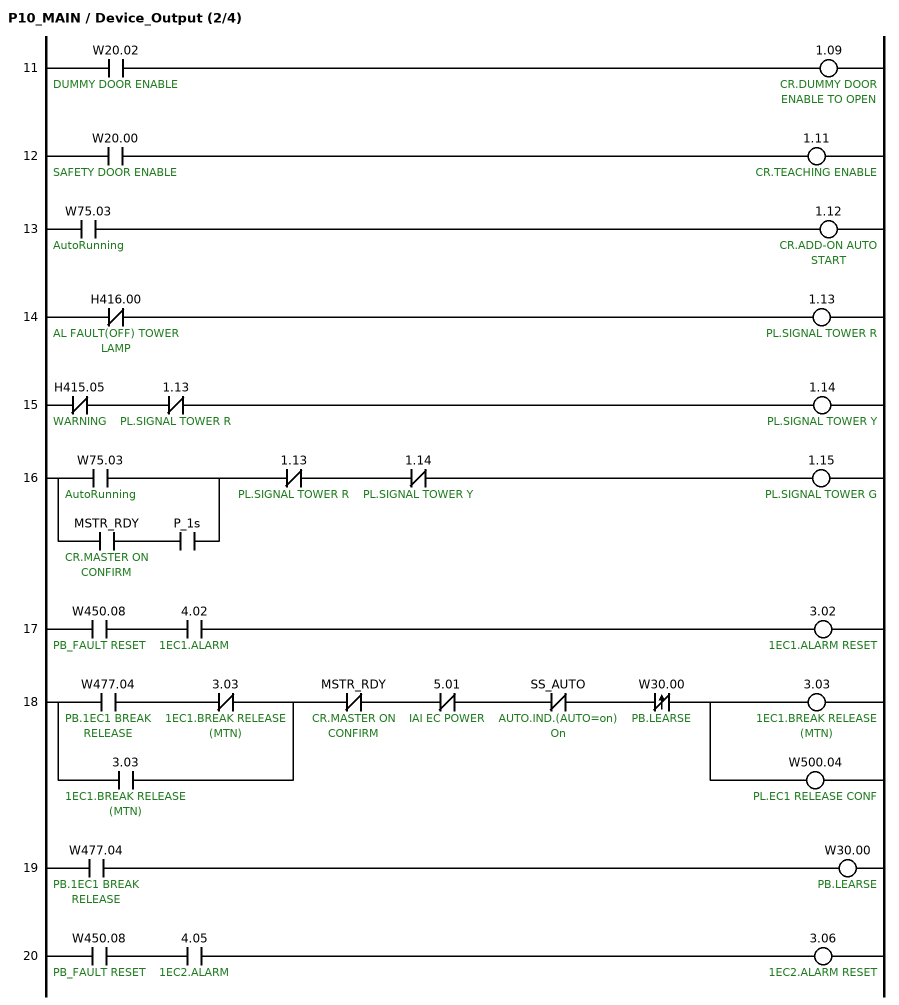
; rung 11
LD W20.02  ; DUMMY DOOR ENABLE
OUT 1.09  ; CR.DUMMY DOOR ENABLE TO OPEN
; rung 12
LD W20.00  ; SAFETY DOOR ENABLE
OUT 1.11  ; CR.TEACHING ENABLE
; rung 13
LD W75.03  ; AutoRunning
OUT 1.12  ; CR.ADD-ON AUTO START
; rung 14
LDNOT H416.00  ; AL FAULT(OFF) TOWER LAMP
OUT 1.13  ; PL.SIGNAL TOWER R
; rung 15
LDNOT H415.05  ; WARNING
ANDNOT 1.13  ; PL.SIGNAL TOWER R
OUT 1.14  ; PL.SIGNAL TOWER Y
; rung 16
LD W75.03  ; AutoRunning
LD MSTR_RDY  ; CR.MASTER ON CONFIRM
AND P_1s
ORLD
ANDNOT 1.13  ; PL.SIGNAL TOWER R
ANDNOT 1.14  ; PL.SIGNAL TOWER Y
OUT 1.15  ; PL.SIGNAL TOWER G
; rung 17
LD W450.08  ; PB_FAULT RESET
AND 4.02  ; 1EC1.ALARM
OUT 3.02  ; 1EC1.ALARM RESET
; rung 18
LD W477.04  ; PB.1EC1 BREAK RELEASE
ANDNOT 3.03  ; 1EC1.BREAK RELEASE (MTN)
OR 3.03  ; 1EC1.BREAK RELEASE (MTN)
ANDNOT MSTR_RDY  ; CR.MASTER ON CONFIRM
ANDNOT 5.01  ; IAI EC POWER
ANDNOT SS_AUTO  ; AUTO.IND.(AUTO=on) On
@ANDNOT W30.00  ; PB.LEARSE
OUT 3.03  ; 1EC1.BREAK RELEASE (MTN)
OUT W500.04  ; PL.EC1 RELEASE CONF
; rung 19
LD W477.04  ; PB.1EC1 BREAK RELEASE
OUT W30.00  ; PB.LEARSE
; rung 20
LD W450.08  ; PB_FAULT RESET
AND 4.05  ; 1EC2.ALARM
OUT 3.06  ; 1EC2.ALARM RESET

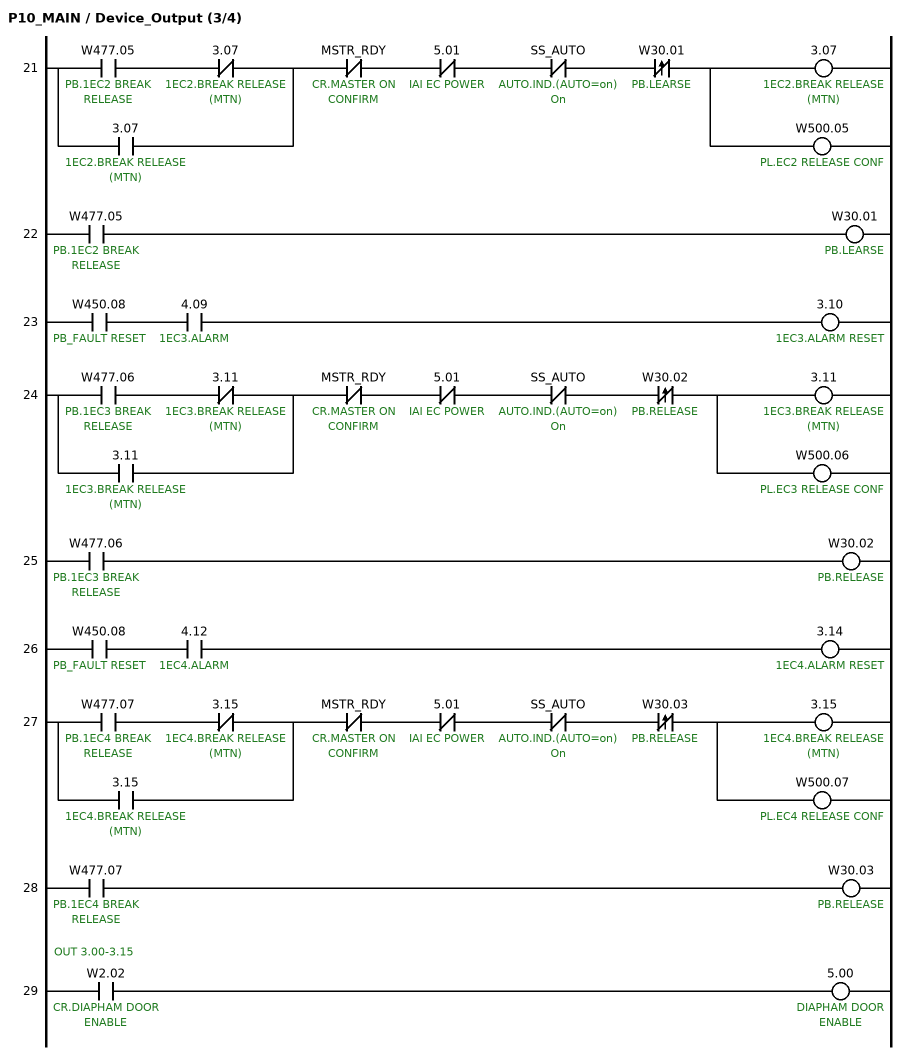
; rung 21
LD W477.05  ; PB.1EC2 BREAK RELEASE
ANDNOT 3.07  ; 1EC2.BREAK RELEASE (MTN)
OR 3.07  ; 1EC2.BREAK RELEASE (MTN)
ANDNOT MSTR_RDY  ; CR.MASTER ON CONFIRM
ANDNOT 5.01  ; IAI EC POWER
ANDNOT SS_AUTO  ; AUTO.IND.(AUTO=on) On
@ANDNOT W30.01  ; PB.LEARSE
OUT 3.07  ; 1EC2.BREAK RELEASE (MTN)
OUT W500.05  ; PL.EC2 RELEASE CONF
; rung 22
LD W477.05  ; PB.1EC2 BREAK RELEASE
OUT W30.01  ; PB.LEARSE
; rung 23
LD W450.08  ; PB_FAULT RESET
AND 4.09  ; 1EC3.ALARM
OUT 3.10  ; 1EC3.ALARM RESET
; rung 24
LD W477.06  ; PB.1EC3 BREAK RELEASE
ANDNOT 3.11  ; 1EC3.BREAK RELEASE (MTN)
OR 3.11  ; 1EC3.BREAK RELEASE (MTN)
ANDNOT MSTR_RDY  ; CR.MASTER ON CONFIRM
ANDNOT 5.01  ; IAI EC POWER
ANDNOT SS_AUTO  ; AUTO.IND.(AUTO=on) On
@ANDNOT W30.02  ; PB.RELEASE
OUT 3.11  ; 1EC3.BREAK RELEASE (MTN)
OUT W500.06  ; PL.EC3 RELEASE CONF
; rung 25
LD W477.06  ; PB.1EC3 BREAK RELEASE
OUT W30.02  ; PB.RELEASE
; rung 26
LD W450.08  ; PB_FAULT RESET
AND 4.12  ; 1EC4.ALARM
OUT 3.14  ; 1EC4.ALARM RESET
; rung 27
LD W477.07  ; PB.1EC4 BREAK RELEASE
ANDNOT 3.15  ; 1EC4.BREAK RELEASE (MTN)
OR 3.15  ; 1EC4.BREAK RELEASE (MTN)
ANDNOT MSTR_RDY  ; CR.MASTER ON CONFIRM
ANDNOT 5.01  ; IAI EC POWER
ANDNOT SS_AUTO  ; AUTO.IND.(AUTO=on) On
@ANDNOT W30.03  ; PB.RELEASE
OUT 3.15  ; 1EC4.BREAK RELEASE (MTN)
OUT W500.07  ; PL.EC4 RELEASE CONF
; rung 28
LD W477.07  ; PB.1EC4 BREAK RELEASE
OUT W30.03  ; PB.RELEASE
; rung 29: OUT 3.00-3.15
LD W2.02  ; CR.DIAPHAM DOOR ENABLE
OUT 5.00  ; DIAPHAM DOOR ENABLE

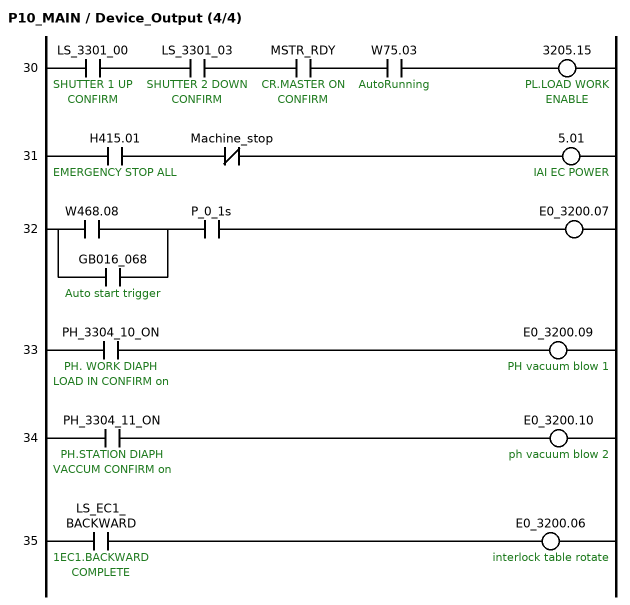
; rung 30
LD LS_3301_00  ; SHUTTER 1 UP CONFIRM
AND LS_3301_03  ; SHUTTER 2 DOWN CONFIRM
AND MSTR_RDY  ; CR.MASTER ON CONFIRM
AND W75.03  ; AutoRunning
OUT 3205.15  ; PL.LOAD WORK ENABLE
; rung 31
LD H415.01  ; EMERGENCY STOP ALL
ANDNOT Machine_stop
OUT 5.01  ; IAI EC POWER
; rung 32
LD W468.08
OR GB016_068  ; Auto start trigger
AND P_0_1s
OUT E0_3200.07
; rung 33
LD PH_3304_10_ON  ; PH. WORK DIAPH LOAD IN CONFIRM on
OUT E0_3200.09  ; PH vacuum blow 1
; rung 34
LD PH_3304_11_ON  ; PH.STATION DIAPH VACCUM CONFIRM on
OUT E0_3200.10  ; ph vacuum blow 2
; rung 35
LD LS_EC1_BACKWARD  ; 1EC1.BACKWARD COMPLETE
OUT E0_3200.06  ; interlock table rotate

### Section LS_ASSIS

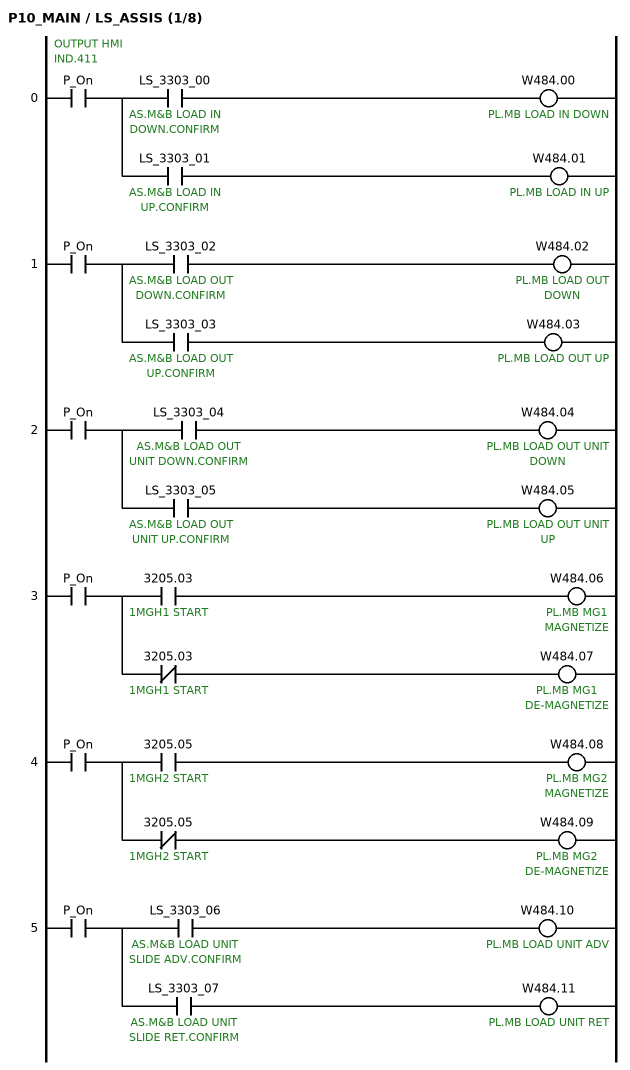
; rung 0: OUTPUT HMI / IND.411
LD P_On
OUT TR0
AND LS_3303_00  ; AS.M&B LOAD IN DOWN.CONFIRM
OUT W484.00  ; PL.MB LOAD IN DOWN
LD TR0
AND LS_3303_01  ; AS.M&B LOAD IN UP.CONFIRM
OUT W484.01  ; PL.MB LOAD IN UP
; rung 1
LD P_On
OUT TR0
AND LS_3303_02  ; AS.M&B LOAD OUT DOWN.CONFIRM
OUT W484.02  ; PL.MB LOAD OUT DOWN
LD TR0
AND LS_3303_03  ; AS.M&B LOAD OUT UP.CONFIRM
OUT W484.03  ; PL.MB LOAD OUT UP
; rung 2
LD P_On
OUT TR0
AND LS_3303_04  ; AS.M&B LOAD OUT UNIT DOWN.CONFIRM
OUT W484.04  ; PL.MB LOAD OUT UNIT DOWN
LD TR0
AND LS_3303_05  ; AS.M&B LOAD OUT UNIT UP.CONFIRM
OUT W484.05  ; PL.MB LOAD OUT UNIT UP
; rung 3
LD P_On
OUT TR0
AND 3205.03  ; 1MGH1 START
OUT W484.06  ; PL.MB MG1 MAGNETIZE
LD TR0
ANDNOT 3205.03  ; 1MGH1 START
OUT W484.07  ; PL.MB MG1 DE-MAGNETIZE
; rung 4
LD P_On
OUT TR0
AND 3205.05  ; 1MGH2 START
OUT W484.08  ; PL.MB MG2 MAGNETIZE
LD TR0
ANDNOT 3205.05  ; 1MGH2 START
OUT W484.09  ; PL.MB MG2 DE-MAGNETIZE
; rung 5
LD P_On
OUT TR0
AND LS_3303_06  ; AS.M&B LOAD UNIT SLIDE ADV.CONFIRM
OUT W484.10  ; PL.MB LOAD UNIT ADV
LD TR0
AND LS_3303_07  ; AS.M&B LOAD UNIT SLIDE RET.CONFIRM
OUT W484.11  ; PL.MB LOAD UNIT RET

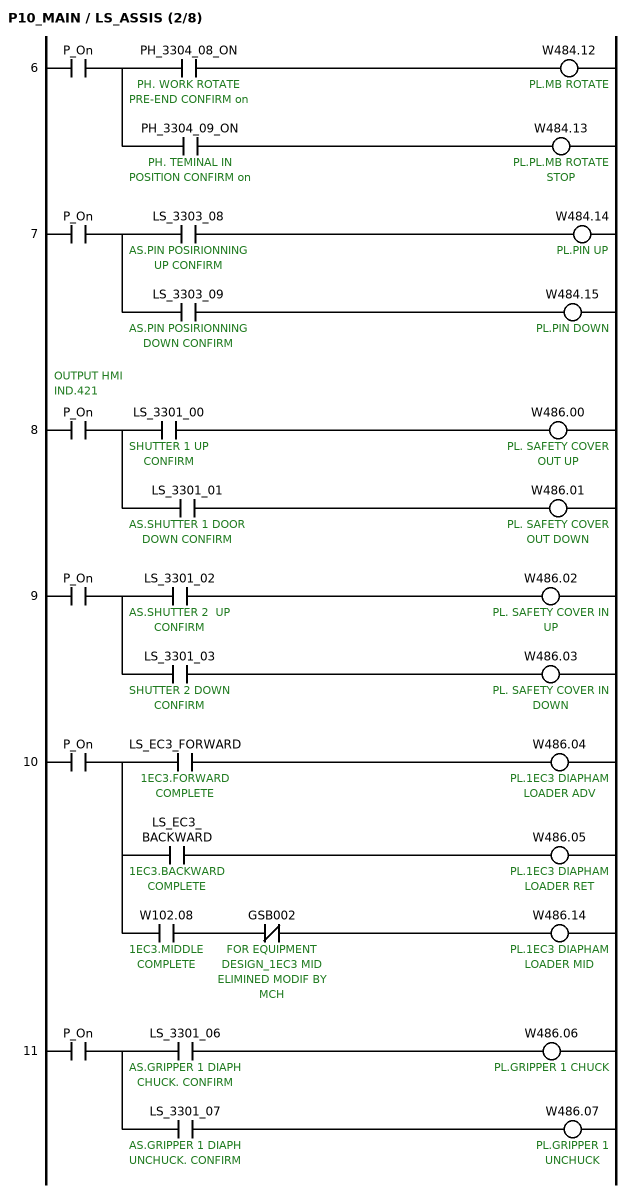
; rung 6
LD P_On
OUT TR0
AND PH_3304_08_ON  ; PH. WORK ROTATE PRE-END CONFIRM on
OUT W484.12  ; PL.MB ROTATE
LD TR0
AND PH_3304_09_ON  ; PH. TEMINAL IN POSITION CONFIRM on
OUT W484.13  ; PL.PL.MB ROTATE STOP
; rung 7
LD P_On
OUT TR0
AND LS_3303_08  ; AS.PIN POSIRIONNING UP CONFIRM
OUT W484.14  ; PL.PIN UP
LD TR0
AND LS_3303_09  ; AS.PIN POSIRIONNING DOWN CONFIRM
OUT W484.15  ; PL.PIN DOWN
; rung 8: OUTPUT HMI / IND.421
LD P_On
OUT TR0
AND LS_3301_00  ; SHUTTER 1 UP CONFIRM
OUT W486.00  ; PL. SAFETY COVER OUT UP
LD TR0
AND LS_3301_01  ; AS.SHUTTER 1 DOOR DOWN CONFIRM
OUT W486.01  ; PL. SAFETY COVER OUT DOWN
; rung 9
LD P_On
OUT TR0
AND LS_3301_02  ; AS.SHUTTER 2  UP CONFIRM
OUT W486.02  ; PL. SAFETY COVER IN UP
LD TR0
AND LS_3301_03  ; SHUTTER 2 DOWN CONFIRM
OUT W486.03  ; PL. SAFETY COVER IN DOWN
; rung 10
LD P_On
OUT TR0
AND LS_EC3_FORWARD  ; 1EC3.FORWARD COMPLETE
OUT W486.04  ; PL.1EC3 DIAPHAM LOADER ADV
LD TR0
AND LS_EC3_BACKWARD  ; 1EC3.BACKWARD COMPLETE
OUT W486.05  ; PL.1EC3 DIAPHAM LOADER RET
LD TR0
AND W102.08  ; 1EC3.MIDDLE COMPLETE
ANDNOT GSB002  ; FOR EQUIPMENT DESIGN_1EC3 MID ELIMINED MODIF BY MCH
OUT W486.14  ; PL.1EC3 DIAPHAM LOADER MID
; rung 11
LD P_On
OUT TR0
AND LS_3301_06  ; AS.GRIPPER 1 DIAPH CHUCK. CONFIRM
OUT W486.06  ; PL.GRIPPER 1 CHUCK
LD TR0
AND LS_3301_07  ; AS.GRIPPER 1 DIAPH UNCHUCK. CONFIRM
OUT W486.07  ; PL.GRIPPER 1 UNCHUCK

